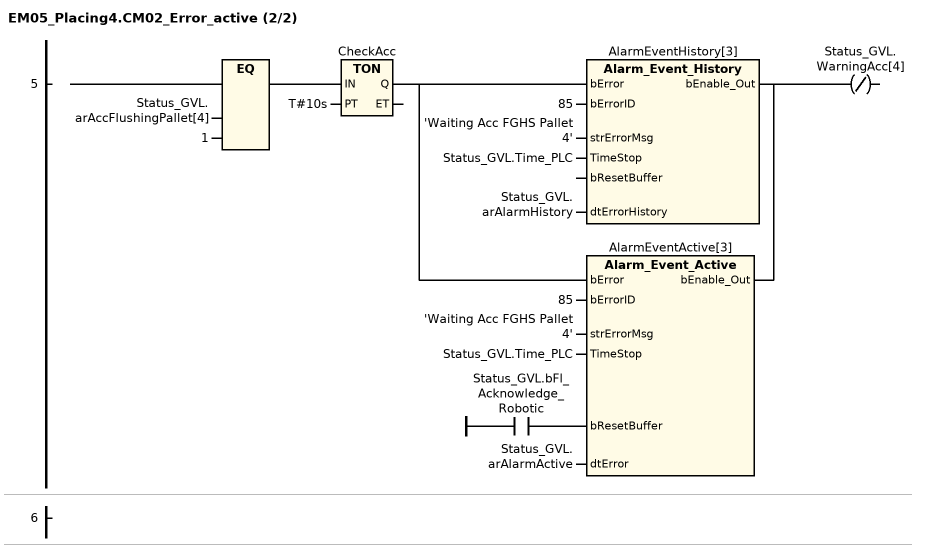
// NETWORK 5
CheckAcc(IN := Status_GVL.arAccFlushingPallet[4] = 1, PT := T#10s); // TON
AlarmEventHistory[3](
    bError := CheckAcc.Q,
    bErrorID := 85,
    strErrorMsg := 'Waiting Acc FGHS Pallet 4',
    TimeStop := Status_GVL.Time_PLC,
    dtErrorHistory := Status_GVL.arAlarmHistory); // Alarm_Event_History
AlarmEventActive[3](
    bError := CheckAcc.Q,
    bErrorID := 85,
    strErrorMsg := 'Waiting Acc FGHS Pallet 4',
    TimeStop := Status_GVL.Time_PLC,
    bResetBuffer := Status_GVL.bFl_Acknowledge_Robotic,
    dtError := Status_GVL.arAlarmActive); // Alarm_Event_Active
Status_GVL.WarningAcc[4] := NOT (AlarmEventHistory[3].bEnable_Out OR AlarmEventActive[3].bEnable_Out);

// NETWORK 6
END_ACTION

ACTION CM03_Output_active:
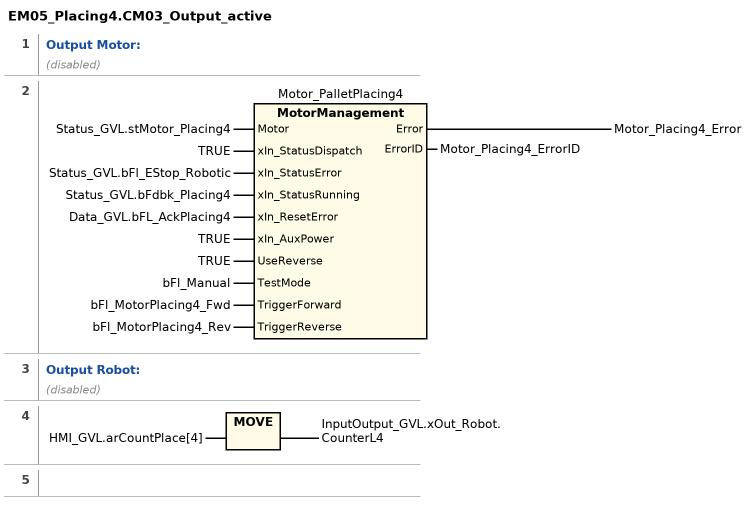
// NETWORK 1 (disabled)
// label: Output Motor

// NETWORK 2
Motor_PalletPlacing4(
    Motor := Status_GVL.stMotor_Placing4,
    xIn_StatusDispatch := TRUE,
    xIn_StatusError := Status_GVL.bFl_EStop_Robotic,
    xIn_StatusRunning := Status_GVL.bFdbk_Placing4,
    xIn_ResetError := Data_GVL.bFL_AckPlacing4,
    xIn_AuxPower := TRUE,
    UseReverse := TRUE,
    TestMode := bFl_Manual,
    TriggerForward := bFl_MotorPlacing4_Fwd,
    TriggerReverse := bFl_MotorPlacing4_Rev,
    ErrorID => Motor_Placing4_ErrorID); // MotorManagement
Motor_Placing4_Error := Motor_PalletPlacing4.Error;

// NETWORK 3 (disabled)
// label: Output Robot

// NETWORK 4
InputOutput_GVL.xOut_Robot.CounterL4 := HMI_GVL.arCountPlace[4];

// NETWORK 5
END_ACTION

ACTION CM04_Running_active:
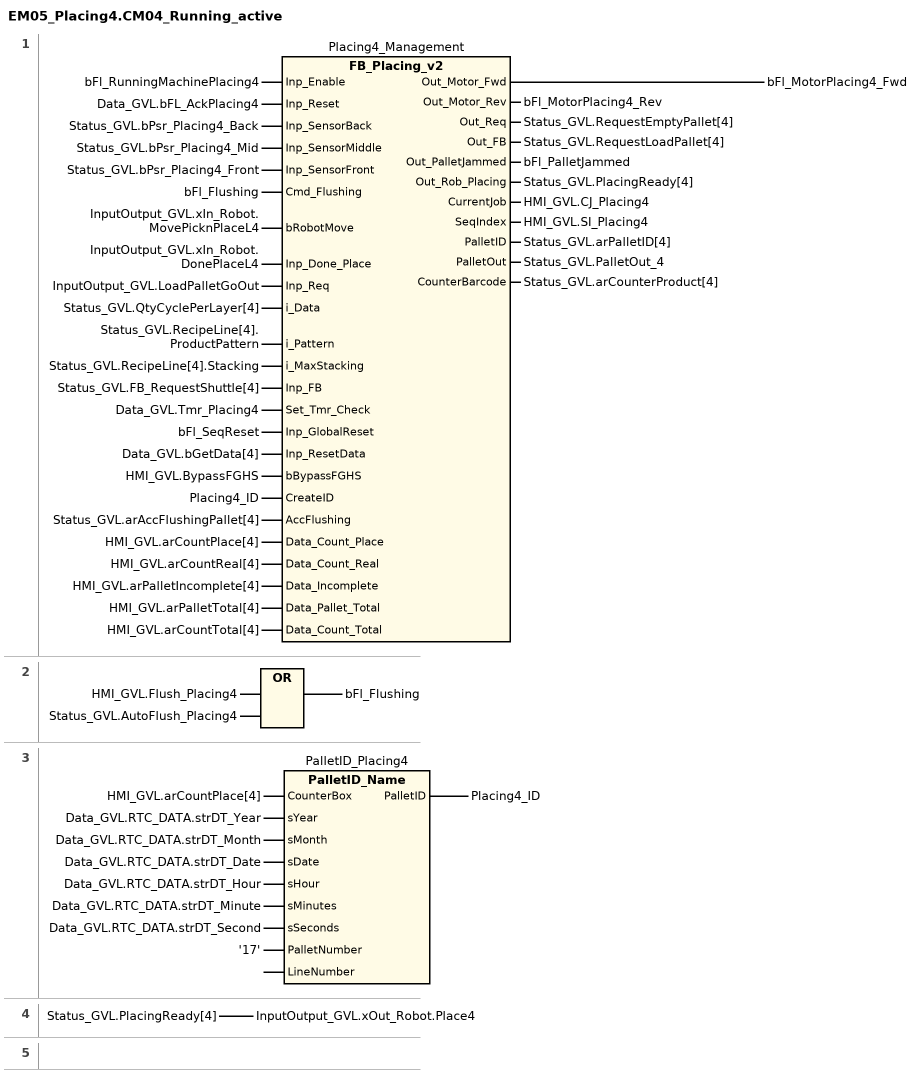
// NETWORK 1
Placing4_Management(
    Inp_Enable := bFl_RunningMachinePlacing4,
    Inp_Reset := Data_GVL.bFL_AckPlacing4,
    Inp_SensorBack := Status_GVL.bPsr_Placing4_Back,
    Inp_SensorMiddle := Status_GVL.bPsr_Placing4_Mid,
    Inp_SensorFront := Status_GVL.bPsr_Placing4_Front,
    Cmd_Flushing := bFl_Flushing,
    bRobotMove := InputOutput_GVL.xIn_Robot.MovePicknPlaceL4,
    Inp_Done_Place := InputOutput_GVL.xIn_Robot.DonePlaceL4,
    Inp_Req := InputOutput_GVL.LoadPalletGoOut,
    i_Data := Status_GVL.QtyCyclePerLayer[4],
    i_Pattern := Status_GVL.RecipeLine[4].ProductPattern,
    i_MaxStacking := Status_GVL.RecipeLine[4].Stacking,
    Inp_FB := Status_GVL.FB_RequestShuttle[4],
    Set_Tmr_Check := Data_GVL.Tmr_Placing4,
    Inp_GlobalReset := bFl_SeqReset,
    Inp_ResetData := Data_GVL.bGetData[4],
    bBypassFGHS := HMI_GVL.BypassFGHS,
    CreateID := Placing4_ID,
    AccFlushing := Status_GVL.arAccFlushingPallet[4],
    Data_Count_Place := HMI_GVL.arCountPlace[4],
    Data_Count_Real := HMI_GVL.arCountReal[4],
    Data_Incomplete := HMI_GVL.arPalletIncomplete[4],
    Data_Pallet_Total := HMI_GVL.arPalletTotal[4],
    Data_Count_Total := HMI_GVL.arCountTotal[4],
    Out_Motor_Rev => bFl_MotorPlacing4_Rev,
    Out_Req => Status_GVL.RequestEmptyPallet[4],
    Out_FB => Status_GVL.RequestLoadPallet[4],
    Out_PalletJammed => bFl_PalletJammed,
    Out_Rob_Placing => Status_GVL.PlacingReady[4],
    CurrentJob => HMI_GVL.CJ_Placing4,
    SeqIndex => HMI_GVL.SI_Placing4,
    PalletID => Status_GVL.arPalletID[4],
    PalletOut => Status_GVL.PalletOut_4,
    CounterBarcode => Status_GVL.arCounterProduct[4]); // FB_Placing_v2
bFl_MotorPlacing4_Fwd := Placing4_Management.Out_Motor_Fwd;

// NETWORK 2
bFl_Flushing := HMI_GVL.Flush_Placing4 OR Status_GVL.AutoFlush_Placing4;

// NETWORK 3
PalletID_Placing4(
    CounterBox := HMI_GVL.arCountPlace[4],
    sYear := Data_GVL.RTC_DATA.strDT_Year,
    sMonth := Data_GVL.RTC_DATA.strDT_Month,
    sDate := Data_GVL.RTC_DATA.strDT_Date,
    sHour := Data_GVL.RTC_DATA.strDT_Hour,
    sMinutes := Data_GVL.RTC_DATA.strDT_Minute,
    sSeconds := Data_GVL.RTC_DATA.strDT_Second,
    PalletNumber := '17'); // PalletID_Name
Placing4_ID := PalletID_Placing4.PalletID;

// NETWORK 4
InputOutput_GVL.xOut_Robot.Place4 := Status_GVL.PlacingReady[4];

// NETWORK 5
END_ACTION

ACTION UP01_Backbone_active:
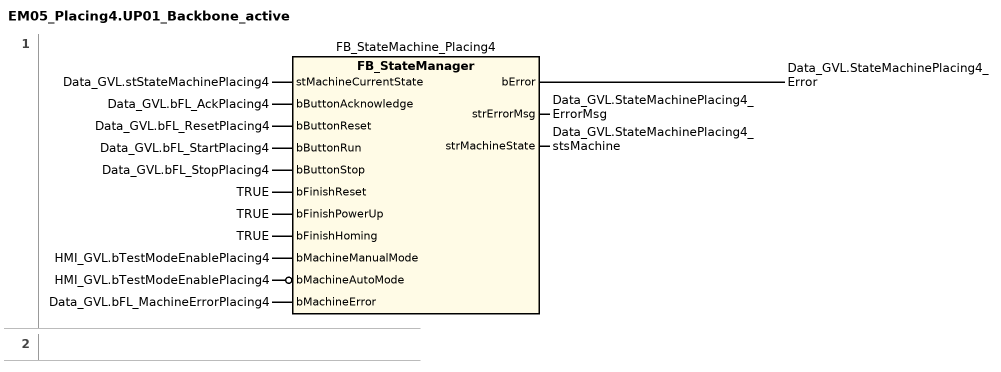
// NETWORK 1
FB_StateMachine_Placing4(
    stMachineCurrentState := Data_GVL.stStateMachinePlacing4,
    bButtonAcknowledge := Data_GVL.bFL_AckPlacing4,
    bButtonReset := Data_GVL.bFL_ResetPlacing4,
    bButtonRun := Data_GVL.bFL_StartPlacing4,
    bButtonStop := Data_GVL.bFL_StopPlacing4,
    bFinishReset := TRUE,
    bFinishPowerUp := TRUE,
    bFinishHoming := TRUE,
    bMachineManualMode := HMI_GVL.bTestModeEnablePlacing4,
    bMachineAutoMode := NOT HMI_GVL.bTestModeEnablePlacing4,
    bMachineError := Data_GVL.bFL_MachineErrorPlacing4,
    strErrorMsg => Data_GVL.StateMachinePlacing4_ErrorMsg,
    strMachineState => Data_GVL.StateMachinePlacing4_stsMachine); // FB_StateManager
Data_GVL.StateMachinePlacing4_Error := FB_StateMachine_Placing4.bError;

// NETWORK 2
END_ACTION

END_PROGRAM

// ---- POUs/S01_Robot/EM06_Picking.TcPOU
PROGRAM EM06_Picking
VAR
	
	//Backbone
	FB_StateMachine_Picking			: FB_StateManager;
	bFl_RunningMachinePicking		: BOOL;
	bFl_SeqReset					: BOOL;
	bFl_Manual						: BOOL;
	CheckStatusPicking				: checkstatus;
	AlarmEventHistory				: ARRAY[1..20] OF Alarm_Event_History;
	ProductFound					: ARRAY [1..4] OF BOOL;
	
	//Motor
	Motor_BoxPicking				: MotorManagement;
	bFl_MotorPicking				: BOOL;
	Motor_Picking_Error				: BOOL;
	Motor_Picking_ErrorID			: UINT;
	
	//Pneumatic
	Pneumatic_GapMaker				: Pneumatic_2Coil_Management;
	bFl_GapMaker_Rtc				: BOOL;
	bFl_GapMaker_Adv				: BOOL;
	Pneu_GapMaker_Error				: BOOL;	
	Pneu_GapMaker_ErrorMsg			: STRING;
	
	Pneumatic_Centering				: Pneumatic_1Coil_Management;
	bFl_Centering					: BOOL;
	Pneu_Centering_Error			: BOOL;	
	Pneu_Centering_ErrorMsg			: STRING;
	
	//Picking
	Picking							: FB_Picking;
	
	//Barcode Reader
	bFl_BarcodeChecked				: BOOL;
	bFl_TriggerBarcode				: BOOL;
	bFl_DoneRead_Barcode_Picking	: ARRAY [1..4] OF BOOL;
	bFl_GoodRead_Barcode_Picking	: ARRAY [1..4] OF BOOL;
	bFl_BadRead_Barcode_Picking		: ARRAY [1..4] OF BOOL;
	BarcodeInspection				: FB_BarcodeInspection;
	BarcodeReader_Picking1			: DM_Connect;
	BarcodeReader_Picking2			: DM_Connect;
	BarcodeReader_Picking3			: DM_Connect;
	BarcodeReader_Picking4			: DM_Connect;
	DataBarcode_Picking1			: STRING;
	DataBarcode_Picking2			: STRING;
	DataBarcode_Picking3			: STRING;
	DataBarcode_Picking4			: STRING;
	Barcode1_Error					: BOOL;
	Barcode2_Error					: BOOL;
	Barcode3_Error					: BOOL;
	Barcode4_Error					: BOOL;
	TestRun							: BOOL;
	TestTrigger						: BOOL;
	LEN1							: INT;
	POS1							: INT;
	POS2							: INT;
	LEN_2							: INT;
	LinkUp							: STRING(255);
	RotatePicking					: RotatePick;
	DonePick						: BOOL;
	bFL_Safety						: BOOL;
	AutoReset						: BOOL;
	TON_Auto						: TON;
	AutoAck							: BOOL;
	AutoRun							: BOOL;
	TOF_Run							: TOF;
	TOF_Reset						: TOF;
	AlarmEventActive				: ARRAY[1..20] OF Alarm_Event_Active;
	RejectMsgList					: RejectMsgHandling;
	bReject							: BOOL;
	RejectID						: INT;
	RejectMsg						: STRING;
	CounterReject					: UINT;
	bRotate							: BOOL;
	BarcodeReader_Picking2B			: DM_Connect;
	Barcode2B_Error					: BOOL;
	DataBarcode_Picking2B			: STRING;
	bFl_DoneRead_Barcode_Picking2B	: BOOL;
	
	BarcodeReader_Picking3B			: DM_Connect;
	Barcode3B_Error					: BOOL;
	DataBarcode_Picking3B			: STRING;
	intRotatePick					: USINT;
END_VAR
VAR // added by the converter: edge detectors and wires of the graphical bodies
    _w1 : BOOL;
END_VAR

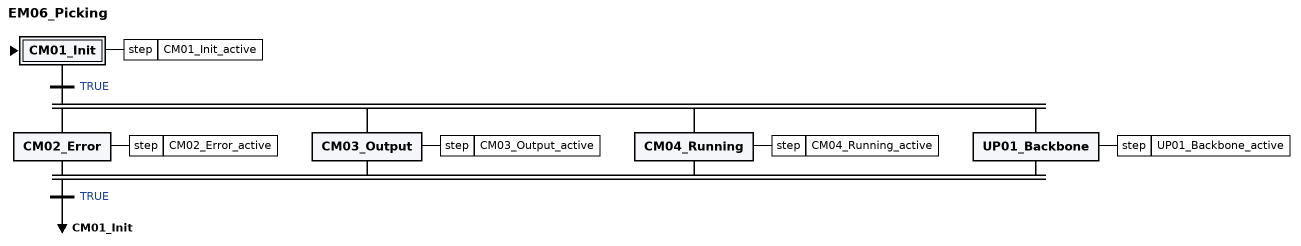
INITIAL_STEP CM01_Init:
    CM01_Init_active(N);  // step action
END_STEP
TRANSITION FROM CM01_Init TO (CM02_Error, CM03_Output, CM04_Running, UP01_Backbone)
    := TRUE;
END_TRANSITION
STEP CM02_Error:
    CM02_Error_active(N);  // step action
END_STEP
STEP CM03_Output:
    CM03_Output_active(N);  // step action
END_STEP
STEP CM04_Running:
    CM04_Running_active(N);  // step action
END_STEP
STEP UP01_Backbone:
    UP01_Backbone_active(N);  // step action
END_STEP
TRANSITION FROM (CM02_Error, CM03_Output, CM04_Running, UP01_Backbone) TO CM01_Init
    := TRUE;
END_TRANSITION

ACTION CM01_Init_active:
Data_GVL.bFL_StartPicking			:= Status_GVL.bFl_RunButton_Robotic OR HMI_GVL.bStartButtonPicking OR HMI_GVL.bAutoStartPicking;
Data_GVL.bFL_StopPicking			:= NOT Status_GVL.bFl_StopButton_Robotic OR HMI_GVL.bStopButtonPicking;
Data_GVL.bFL_ResetPicking			:= Status_GVL.bFl_ResetButton_Robotic OR HMI_GVL.bResetButtonPicking OR HMI_GVL.bAutoResetPicking;
Data_GVL.bFL_AckPicking				:= Status_GVL.bFl_Acknowledge_Robotic OR HMI_GVL.bAcknowledgeButtonPicking OR HMI_GVL.bAutoAcknowledgePicking;
Data_GVL.bFL_AutoManuaModePicking 	:= Status_GVL.bFl_Manual_Robotic OR HMI_GVL.bTestModeEnablePicking;
bFl_RunningMachinePicking			:= Data_GVL.stStateMachinePicking.Running;
bFl_Manual							:= Data_GVL.stStateMachinePicking.ManualMode;
bFl_SeqReset						:= NOT Status_GVL.bFl_EStop_Robotic;
bFL_Safety							:= Status_GVL.bFl_EStop_Robotic AND Status_GVL.bSafety_DoorRobotic AND Status_GVL.bAirPressure_Robotic;



(*=================Convert Timer============================*)
Data_GVL.Tmr_Picking	:= ConvertMilliSecTimeData(HMI_GVL.Tmr_Picking);
Data_GVL.Tmr_Centering	:= ConvertMilliSecTimeData(HMI_GVL.Tmr_Centering);

(*=================Auto Flushing============================*)
//Place1
IF ProductFound[1] AND HMI_GVL.arCountReal[1] > 1 THEN
	Status_GVL.AutoFlush_Placing1	:= TRUE;
ELSE
	Status_GVL.AutoFlush_Placing1	:= FALSE;
END_IF

//Place2
IF ProductFound[2] AND HMI_GVL.arCountReal[2] > 1 THEN
	Status_GVL.AutoFlush_Placing2	:= TRUE;
ELSE
	Status_GVL.AutoFlush_Placing2	:= FALSE;
END_IF

//Place3
IF ProductFound[3] AND HMI_GVL.arCountReal[3] > 1 THEN
	Status_GVL.AutoFlush_Placing3	:= TRUE;
ELSE
	Status_GVL.AutoFlush_Placing3	:= FALSE;
END_IF

//Place4
IF ProductFound[4] AND HMI_GVL.arCountReal[4] > 1 THEN
	Status_GVL.AutoFlush_Placing4	:= TRUE;
ELSE
	Status_GVL.AutoFlush_Placing4	:= FALSE;
END_IF
END_ACTION

ACTION CM02_Error_active:
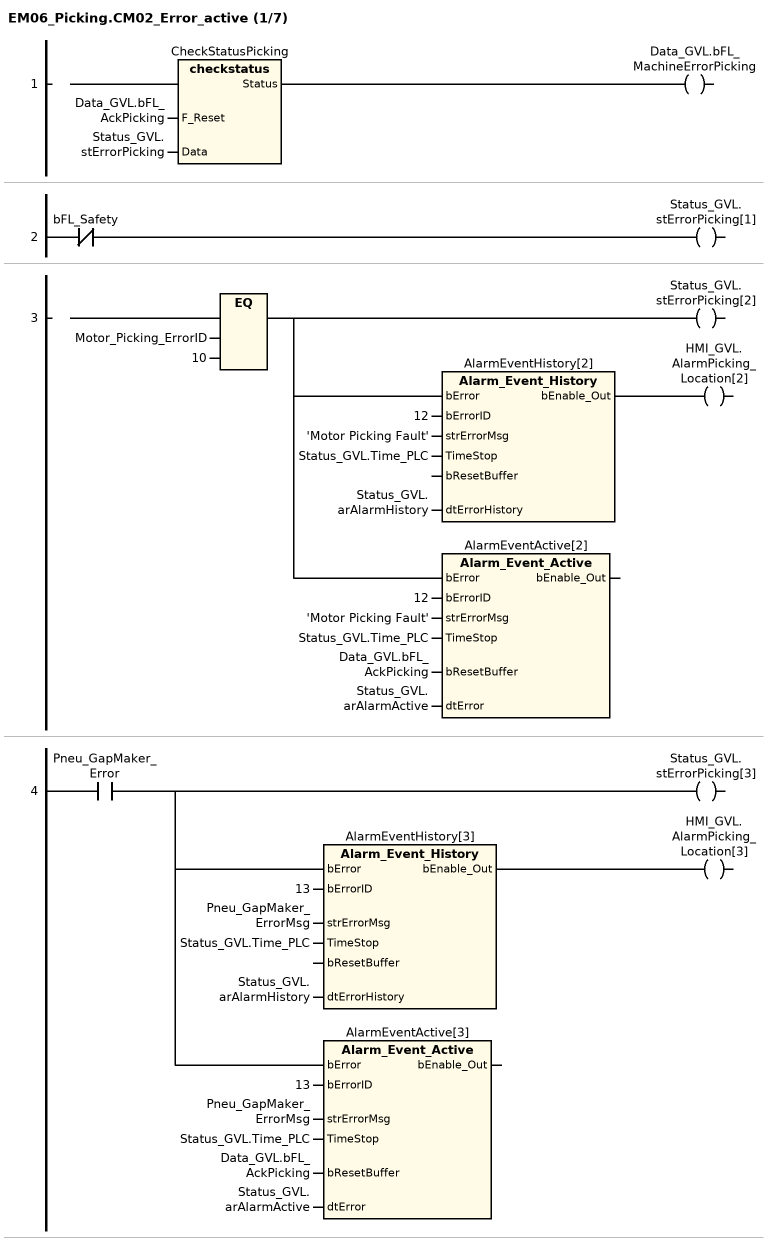
// NETWORK 1
CheckStatusPicking(F_Reset := Data_GVL.bFL_AckPicking, Data := Status_GVL.stErrorPicking); // checkstatus
Data_GVL.bFL_MachineErrorPicking := CheckStatusPicking.Status;

// NETWORK 2
Status_GVL.stErrorPicking[1] := NOT bFL_Safety;

// NETWORK 3
_w1 := Motor_Picking_ErrorID = 10;
Status_GVL.stErrorPicking[2] := _w1;
AlarmEventHistory[2](
    bError := _w1,
    bErrorID := 12,
    strErrorMsg := 'Motor Picking Fault',
    TimeStop := Status_GVL.Time_PLC,
    dtErrorHistory := Status_GVL.arAlarmHistory); // Alarm_Event_History
HMI_GVL.AlarmPicking_Location[2] := AlarmEventHistory[2].bEnable_Out;
AlarmEventActive[2](
    bError := _w1,
    bErrorID := 12,
    strErrorMsg := 'Motor Picking Fault',
    TimeStop := Status_GVL.Time_PLC,
    bResetBuffer := Data_GVL.bFL_AckPicking,
    dtError := Status_GVL.arAlarmActive); // Alarm_Event_Active

// NETWORK 4
Status_GVL.stErrorPicking[3] := Pneu_GapMaker_Error;
AlarmEventHistory[3](
    bError := Pneu_GapMaker_Error,
    bErrorID := 13,
    strErrorMsg := Pneu_GapMaker_ErrorMsg,
    TimeStop := Status_GVL.Time_PLC,
    dtErrorHistory := Status_GVL.arAlarmHistory); // Alarm_Event_History
HMI_GVL.AlarmPicking_Location[3] := AlarmEventHistory[3].bEnable_Out;
AlarmEventActive[3](
    bError := Pneu_GapMaker_Error,
    bErrorID := 13,
    strErrorMsg := Pneu_GapMaker_ErrorMsg,
    TimeStop := Status_GVL.Time_PLC,
    bResetBuffer := Data_GVL.bFL_AckPicking,
    dtError := Status_GVL.arAlarmActive); // Alarm_Event_Active

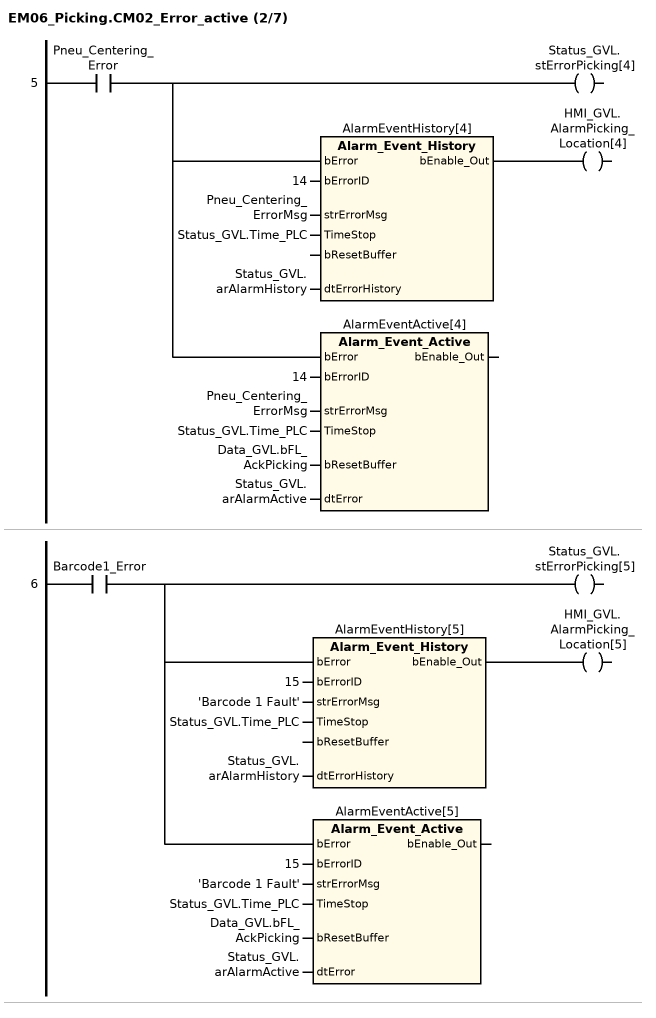
// NETWORK 5
Status_GVL.stErrorPicking[4] := Pneu_Centering_Error;
AlarmEventHistory[4](
    bError := Pneu_Centering_Error,
    bErrorID := 14,
    strErrorMsg := Pneu_Centering_ErrorMsg,
    TimeStop := Status_GVL.Time_PLC,
    dtErrorHistory := Status_GVL.arAlarmHistory); // Alarm_Event_History
HMI_GVL.AlarmPicking_Location[4] := AlarmEventHistory[4].bEnable_Out;
AlarmEventActive[4](
    bError := Pneu_Centering_Error,
    bErrorID := 14,
    strErrorMsg := Pneu_Centering_ErrorMsg,
    TimeStop := Status_GVL.Time_PLC,
    bResetBuffer := Data_GVL.bFL_AckPicking,
    dtError := Status_GVL.arAlarmActive); // Alarm_Event_Active

// NETWORK 6
Status_GVL.stErrorPicking[5] := Barcode1_Error;
AlarmEventHistory[5](
    bError := Barcode1_Error,
    bErrorID := 15,
    strErrorMsg := 'Barcode 1 Fault',
    TimeStop := Status_GVL.Time_PLC,
    dtErrorHistory := Status_GVL.arAlarmHistory); // Alarm_Event_History
HMI_GVL.AlarmPicking_Location[5] := AlarmEventHistory[5].bEnable_Out;
AlarmEventActive[5](
    bError := Barcode1_Error,
    bErrorID := 15,
    strErrorMsg := 'Barcode 1 Fault',
    TimeStop := Status_GVL.Time_PLC,
    bResetBuffer := Data_GVL.bFL_AckPicking,
    dtError := Status_GVL.arAlarmActive); // Alarm_Event_Active

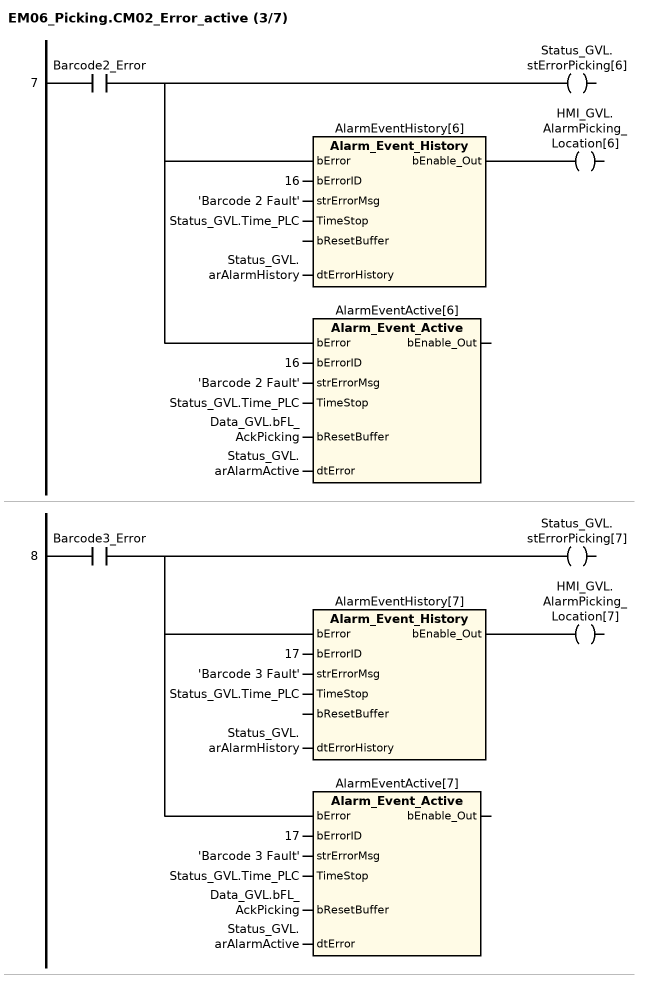
// NETWORK 7
Status_GVL.stErrorPicking[6] := Barcode2_Error;
AlarmEventHistory[6](
    bError := Barcode2_Error,
    bErrorID := 16,
    strErrorMsg := 'Barcode 2 Fault',
    TimeStop := Status_GVL.Time_PLC,
    dtErrorHistory := Status_GVL.arAlarmHistory); // Alarm_Event_History
HMI_GVL.AlarmPicking_Location[6] := AlarmEventHistory[6].bEnable_Out;
AlarmEventActive[6](
    bError := Barcode2_Error,
    bErrorID := 16,
    strErrorMsg := 'Barcode 2 Fault',
    TimeStop := Status_GVL.Time_PLC,
    bResetBuffer := Data_GVL.bFL_AckPicking,
    dtError := Status_GVL.arAlarmActive); // Alarm_Event_Active

// NETWORK 8
Status_GVL.stErrorPicking[7] := Barcode3_Error;
AlarmEventHistory[7](
    bError := Barcode3_Error,
    bErrorID := 17,
    strErrorMsg := 'Barcode 3 Fault',
    TimeStop := Status_GVL.Time_PLC,
    dtErrorHistory := Status_GVL.arAlarmHistory); // Alarm_Event_History
HMI_GVL.AlarmPicking_Location[7] := AlarmEventHistory[7].bEnable_Out;
AlarmEventActive[7](
    bError := Barcode3_Error,
    bErrorID := 17,
    strErrorMsg := 'Barcode 3 Fault',
    TimeStop := Status_GVL.Time_PLC,
    bResetBuffer := Data_GVL.bFL_AckPicking,
    dtError := Status_GVL.arAlarmActive); // Alarm_Event_Active

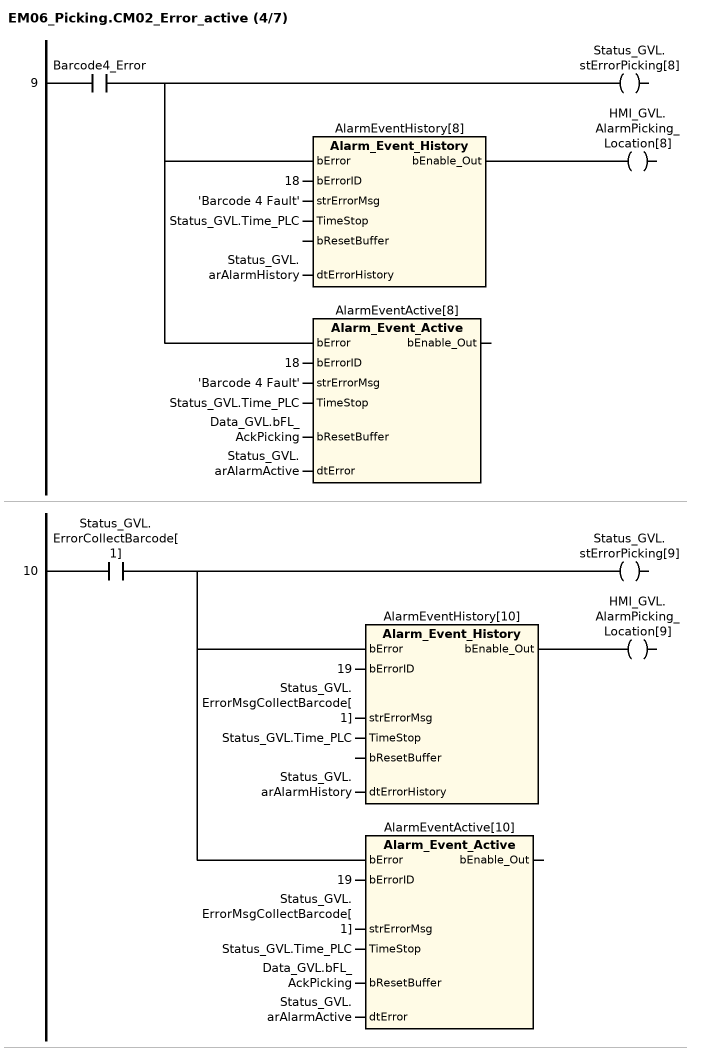
// NETWORK 9
Status_GVL.stErrorPicking[8] := Barcode4_Error;
AlarmEventHistory[8](
    bError := Barcode4_Error,
    bErrorID := 18,
    strErrorMsg := 'Barcode 4 Fault',
    TimeStop := Status_GVL.Time_PLC,
    dtErrorHistory := Status_GVL.arAlarmHistory); // Alarm_Event_History
HMI_GVL.AlarmPicking_Location[8] := AlarmEventHistory[8].bEnable_Out;
AlarmEventActive[8](
    bError := Barcode4_Error,
    bErrorID := 18,
    strErrorMsg := 'Barcode 4 Fault',
    TimeStop := Status_GVL.Time_PLC,
    bResetBuffer := Data_GVL.bFL_AckPicking,
    dtError := Status_GVL.arAlarmActive); // Alarm_Event_Active

// NETWORK 10
Status_GVL.stErrorPicking[9] := Status_GVL.ErrorCollectBarcode[1];
AlarmEventHistory[10](
    bError := Status_GVL.ErrorCollectBarcode[1],
    bErrorID := 19,
    strErrorMsg := Status_GVL.ErrorMsgCollectBarcode[1],
    TimeStop := Status_GVL.Time_PLC,
    dtErrorHistory := Status_GVL.arAlarmHistory); // Alarm_Event_History
HMI_GVL.AlarmPicking_Location[9] := AlarmEventHistory[10].bEnable_Out;
AlarmEventActive[10](
    bError := Status_GVL.ErrorCollectBarcode[1],
    bErrorID := 19,
    strErrorMsg := Status_GVL.ErrorMsgCollectBarcode[1],
    TimeStop := Status_GVL.Time_PLC,
    bResetBuffer := Data_GVL.bFL_AckPicking,
    dtError := Status_GVL.arAlarmActive); // Alarm_Event_Active

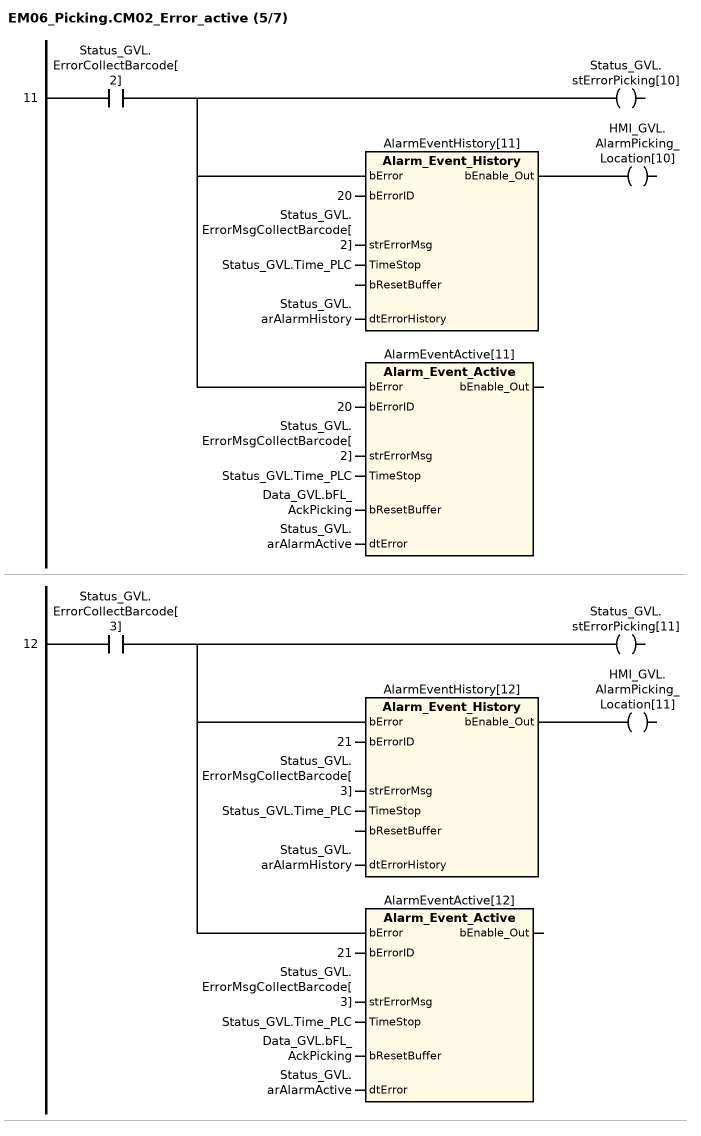
// NETWORK 11
Status_GVL.stErrorPicking[10] := Status_GVL.ErrorCollectBarcode[2];
AlarmEventHistory[11](
    bError := Status_GVL.ErrorCollectBarcode[2],
    bErrorID := 20,
    strErrorMsg := Status_GVL.ErrorMsgCollectBarcode[2],
    TimeStop := Status_GVL.Time_PLC,
    dtErrorHistory := Status_GVL.arAlarmHistory); // Alarm_Event_History
HMI_GVL.AlarmPicking_Location[10] := AlarmEventHistory[11].bEnable_Out;
AlarmEventActive[11](
    bError := Status_GVL.ErrorCollectBarcode[2],
    bErrorID := 20,
    strErrorMsg := Status_GVL.ErrorMsgCollectBarcode[2],
    TimeStop := Status_GVL.Time_PLC,
    bResetBuffer := Data_GVL.bFL_AckPicking,
    dtError := Status_GVL.arAlarmActive); // Alarm_Event_Active

// NETWORK 12
Status_GVL.stErrorPicking[11] := Status_GVL.ErrorCollectBarcode[3];
AlarmEventHistory[12](
    bError := Status_GVL.ErrorCollectBarcode[3],
    bErrorID := 21,
    strErrorMsg := Status_GVL.ErrorMsgCollectBarcode[3],
    TimeStop := Status_GVL.Time_PLC,
    dtErrorHistory := Status_GVL.arAlarmHistory); // Alarm_Event_History
HMI_GVL.AlarmPicking_Location[11] := AlarmEventHistory[12].bEnable_Out;
AlarmEventActive[12](
    bError := Status_GVL.ErrorCollectBarcode[3],
    bErrorID := 21,
    strErrorMsg := Status_GVL.ErrorMsgCollectBarcode[3],
    TimeStop := Status_GVL.Time_PLC,
    bResetBuffer := Data_GVL.bFL_AckPicking,
    dtError := Status_GVL.arAlarmActive); // Alarm_Event_Active

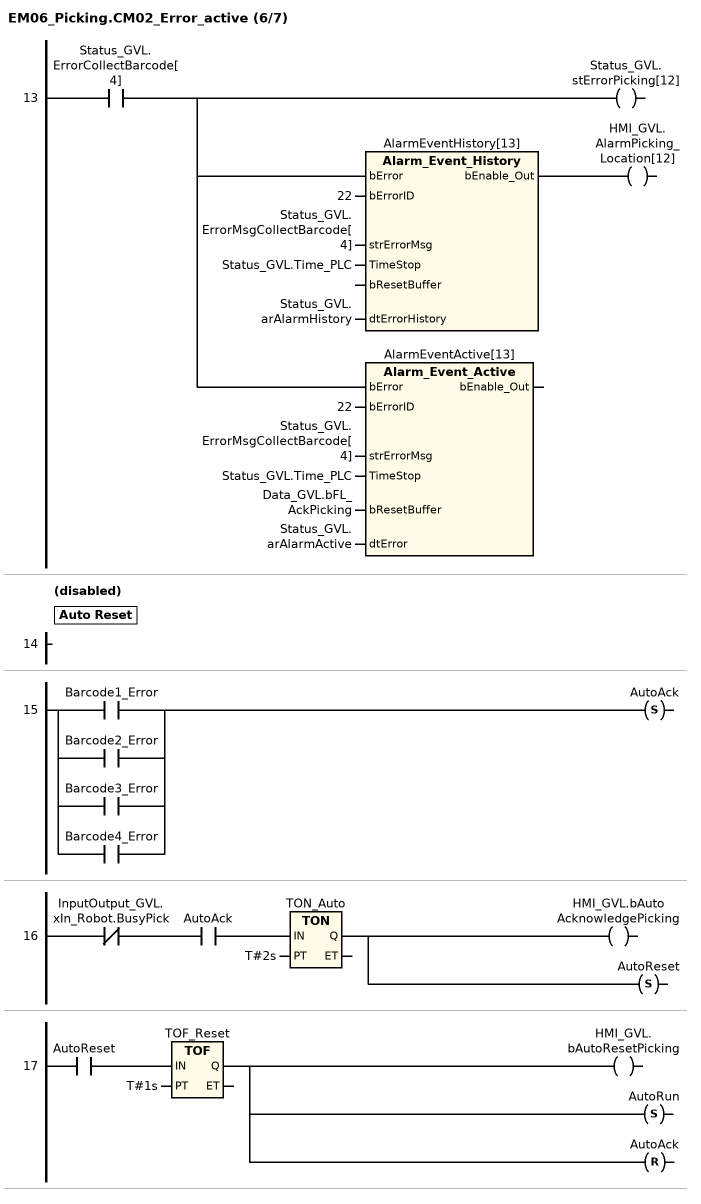
// NETWORK 13
Status_GVL.stErrorPicking[12] := Status_GVL.ErrorCollectBarcode[4];
AlarmEventHistory[13](
    bError := Status_GVL.ErrorCollectBarcode[4],
    bErrorID := 22,
    strErrorMsg := Status_GVL.ErrorMsgCollectBarcode[4],
    TimeStop := Status_GVL.Time_PLC,
    dtErrorHistory := Status_GVL.arAlarmHistory); // Alarm_Event_History
HMI_GVL.AlarmPicking_Location[12] := AlarmEventHistory[13].bEnable_Out;
AlarmEventActive[13](
    bError := Status_GVL.ErrorCollectBarcode[4],
    bErrorID := 22,
    strErrorMsg := Status_GVL.ErrorMsgCollectBarcode[4],
    TimeStop := Status_GVL.Time_PLC,
    bResetBuffer := Data_GVL.bFL_AckPicking,
    dtError := Status_GVL.arAlarmActive); // Alarm_Event_Active

// NETWORK 14 (disabled)
// label: Auto Reset

// NETWORK 15
AutoAck S= Barcode1_Error OR Barcode2_Error OR Barcode3_Error OR Barcode4_Error;

// NETWORK 16
TON_Auto(IN := NOT InputOutput_GVL.xIn_Robot.BusyPick AND AutoAck, PT := T#2s); // TON
HMI_GVL.bAutoAcknowledgePicking := TON_Auto.Q;
AutoReset S= TON_Auto.Q;

// NETWORK 17
TOF_Reset(IN := AutoReset, PT := T#1s); // TOF
HMI_GVL.bAutoResetPicking := TOF_Reset.Q;
AutoRun S= TOF_Reset.Q;
AutoAck R= TOF_Reset.Q;

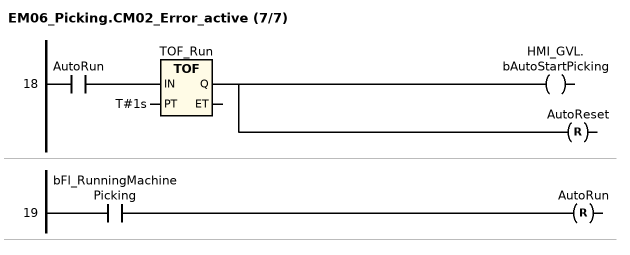
// NETWORK 18
TOF_Run(IN := AutoRun, PT := T#1s); // TOF
HMI_GVL.bAutoStartPicking := TOF_Run.Q;
AutoReset R= TOF_Run.Q;

// NETWORK 19
AutoRun R= bFl_RunningMachinePicking;
END_ACTION

ACTION CM03_Output_active:
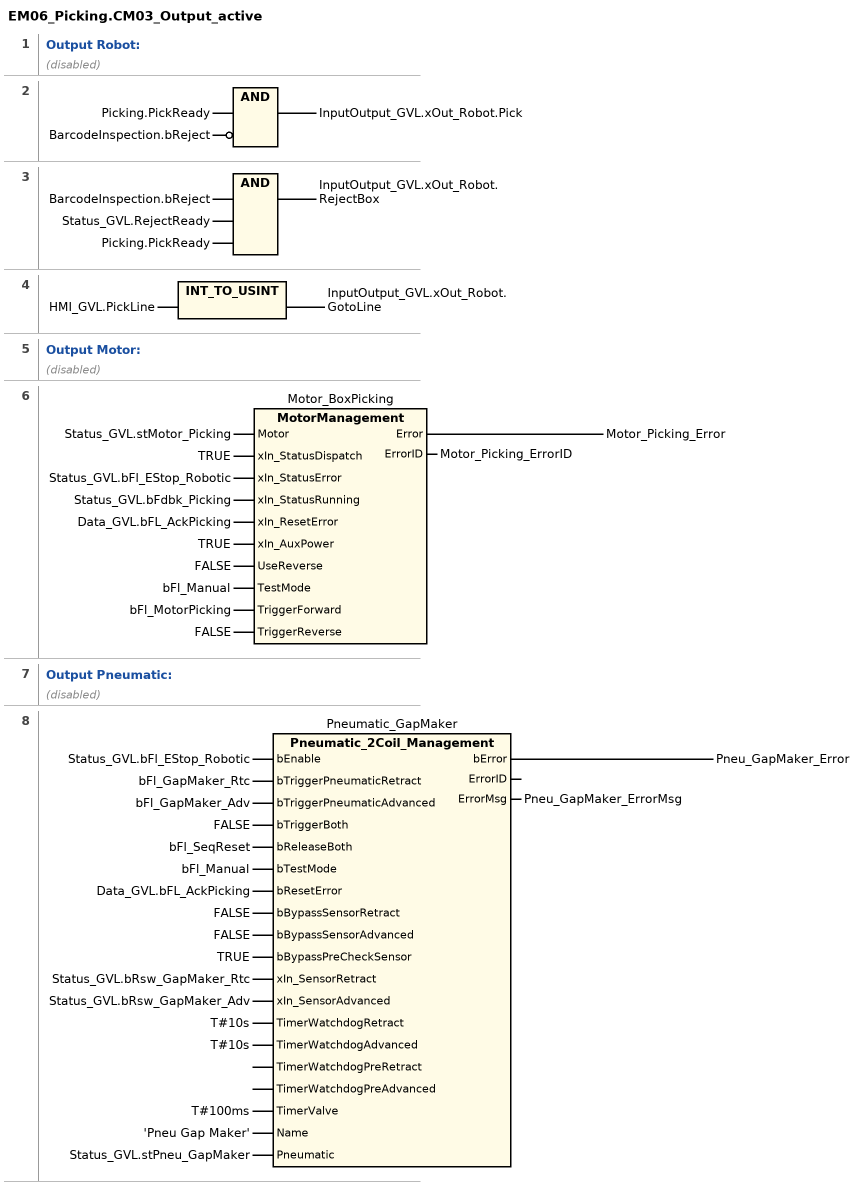
// NETWORK 1 (disabled)
// label: Output Robot

// NETWORK 2
InputOutput_GVL.xOut_Robot.Pick := Picking.PickReady AND NOT BarcodeInspection.bReject;

// NETWORK 3
InputOutput_GVL.xOut_Robot.RejectBox := BarcodeInspection.bReject AND Status_GVL.RejectReady AND Picking.PickReady;

// NETWORK 4
InputOutput_GVL.xOut_Robot.GotoLine := INT_TO_USINT(HMI_GVL.PickLine);

// NETWORK 5 (disabled)
// label: Output Motor

// NETWORK 6
Motor_BoxPicking(
    Motor := Status_GVL.stMotor_Picking,
    xIn_StatusDispatch := TRUE,
    xIn_StatusError := Status_GVL.bFl_EStop_Robotic,
    xIn_StatusRunning := Status_GVL.bFdbk_Picking,
    xIn_ResetError := Data_GVL.bFL_AckPicking,
    xIn_AuxPower := TRUE,
    UseReverse := FALSE,
    TestMode := bFl_Manual,
    TriggerForward := bFl_MotorPicking,
    TriggerReverse := FALSE,
    ErrorID => Motor_Picking_ErrorID); // MotorManagement
Motor_Picking_Error := Motor_BoxPicking.Error;

// NETWORK 7 (disabled)
// label: Output Pneumatic

// NETWORK 8
Pneumatic_GapMaker(
    bEnable := Status_GVL.bFl_EStop_Robotic,
    bTriggerPneumaticRetract := bFl_GapMaker_Rtc,
    bTriggerPneumaticAdvanced := bFl_GapMaker_Adv,
    bTriggerBoth := FALSE,
    bReleaseBoth := bFl_SeqReset,
    bTestMode := bFl_Manual,
    bResetError := Data_GVL.bFL_AckPicking,
    bBypassSensorRetract := FALSE,
    bBypassSensorAdvanced := FALSE,
    bBypassPreCheckSensor := TRUE,
    xIn_SensorRetract := Status_GVL.bRsw_GapMaker_Rtc,
    xIn_SensorAdvanced := Status_GVL.bRsw_GapMaker_Adv,
    TimerWatchdogRetract := T#10s,
    TimerWatchdogAdvanced := T#10s,
    TimerValve := T#100ms,
    Name := 'Pneu Gap Maker',
    Pneumatic := Status_GVL.stPneu_GapMaker,
    ErrorMsg => Pneu_GapMaker_ErrorMsg); // Pneumatic_2Coil_Management
Pneu_GapMaker_Error := Pneumatic_GapMaker.bError;

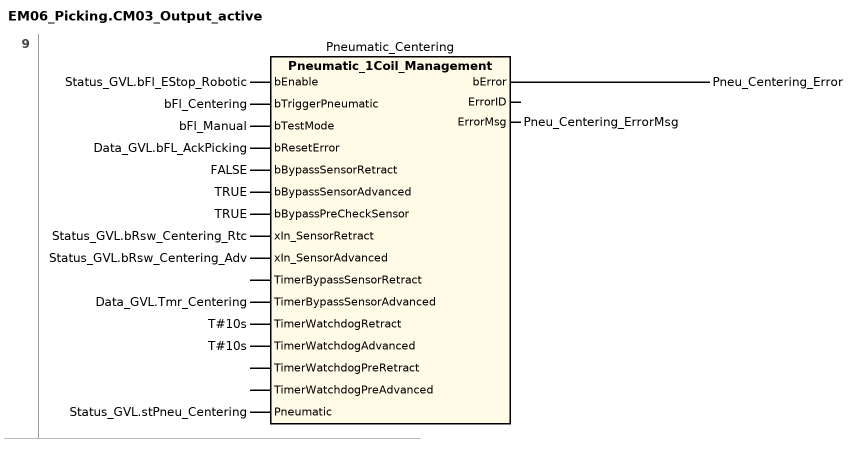
// NETWORK 9
Pneumatic_Centering(
    bEnable := Status_GVL.bFl_EStop_Robotic,
    bTriggerPneumatic := bFl_Centering,
    bTestMode := bFl_Manual,
    bResetError := Data_GVL.bFL_AckPicking,
    bBypassSensorRetract := FALSE,
    bBypassSensorAdvanced := TRUE,
    bBypassPreCheckSensor := TRUE,
    xIn_SensorRetract := Status_GVL.bRsw_Centering_Rtc,
    xIn_SensorAdvanced := Status_GVL.bRsw_Centering_Adv,
    TimerBypassSensorAdvanced := Data_GVL.Tmr_Centering,
    TimerWatchdogRetract := T#10s,
    TimerWatchdogAdvanced := T#10s,
    Pneumatic := Status_GVL.stPneu_Centering,
    ErrorMsg => Pneu_Centering_ErrorMsg); // Pneumatic_1Coil_Management
Pneu_Centering_Error := Pneumatic_Centering.bError;
END_ACTION

ACTION CM04_Running_active:
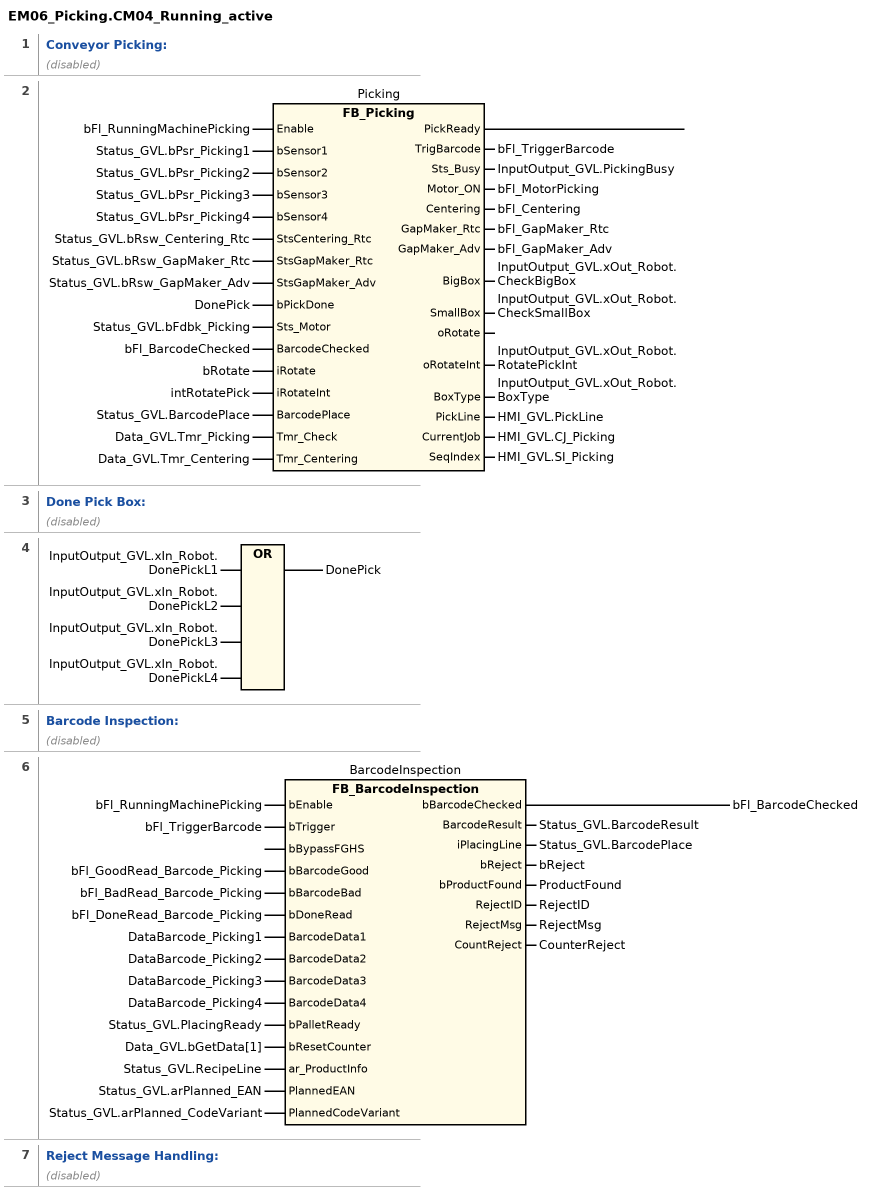
// NETWORK 1 (disabled)
// label: Conveyor Picking

// NETWORK 2
Picking(
    Enable := bFl_RunningMachinePicking,
    bSensor1 := Status_GVL.bPsr_Picking1,
    bSensor2 := Status_GVL.bPsr_Picking2,
    bSensor3 := Status_GVL.bPsr_Picking3,
    bSensor4 := Status_GVL.bPsr_Picking4,
    StsCentering_Rtc := Status_GVL.bRsw_Centering_Rtc,
    StsGapMaker_Rtc := Status_GVL.bRsw_GapMaker_Rtc,
    StsGapMaker_Adv := Status_GVL.bRsw_GapMaker_Adv,
    bPickDone := DonePick,
    Sts_Motor := Status_GVL.bFdbk_Picking,
    BarcodeChecked := bFl_BarcodeChecked,
    iRotate := bRotate,
    iRotateInt := intRotatePick,
    BarcodePlace := Status_GVL.BarcodePlace,
    Tmr_Check := Data_GVL.Tmr_Picking,
    Tmr_Centering := Data_GVL.Tmr_Centering,
    TrigBarcode => bFl_TriggerBarcode,
    Sts_Busy => InputOutput_GVL.PickingBusy,
    Motor_ON => bFl_MotorPicking,
    Centering => bFl_Centering,
    GapMaker_Rtc => bFl_GapMaker_Rtc,
    GapMaker_Adv => bFl_GapMaker_Adv,
    BigBox => InputOutput_GVL.xOut_Robot.CheckBigBox,
    SmallBox => InputOutput_GVL.xOut_Robot.CheckSmallBox,
    oRotateInt => InputOutput_GVL.xOut_Robot.RotatePickInt,
    BoxType => InputOutput_GVL.xOut_Robot.BoxType,
    PickLine => HMI_GVL.PickLine,
    CurrentJob => HMI_GVL.CJ_Picking,
    SeqIndex => HMI_GVL.SI_Picking); // FB_Picking

// NETWORK 3 (disabled)
// label: Done Pick Box

// NETWORK 4
DonePick := InputOutput_GVL.xIn_Robot.DonePickL1 OR InputOutput_GVL.xIn_Robot.DonePickL2 OR InputOutput_GVL.xIn_Robot.DonePickL3 OR InputOutput_GVL.xIn_Robot.DonePickL4;

// NETWORK 5 (disabled)
// label: Barcode Inspection

// NETWORK 6
BarcodeInspection(
    bEnable := bFl_RunningMachinePicking,
    bTrigger := bFl_TriggerBarcode,
    bBarcodeGood := bFl_GoodRead_Barcode_Picking,
    bBarcodeBad := bFl_BadRead_Barcode_Picking,
    bDoneRead := bFl_DoneRead_Barcode_Picking,
    BarcodeData1 := DataBarcode_Picking1,
    BarcodeData2 := DataBarcode_Picking2,
    BarcodeData3 := DataBarcode_Picking3,
    BarcodeData4 := DataBarcode_Picking4,
    bPalletReady := Status_GVL.PlacingReady,
    bResetCounter := Data_GVL.bGetData[1],
    ar_ProductInfo := Status_GVL.RecipeLine,
    PlannedEAN := Status_GVL.arPlanned_EAN,
    PlannedCodeVariant := Status_GVL.arPlanned_CodeVariant,
    BarcodeResult => Status_GVL.BarcodeResult,
    iPlacingLine => Status_GVL.BarcodePlace,
    bReject => bReject,
    bProductFound => ProductFound,
    RejectID => RejectID,
    RejectMsg => RejectMsg,
    CountReject => CounterReject); // FB_BarcodeInspection
bFl_BarcodeChecked := BarcodeInspection.bBarcodeChecked;

// NETWORK 7 (disabled)
// label: Reject Message Handling

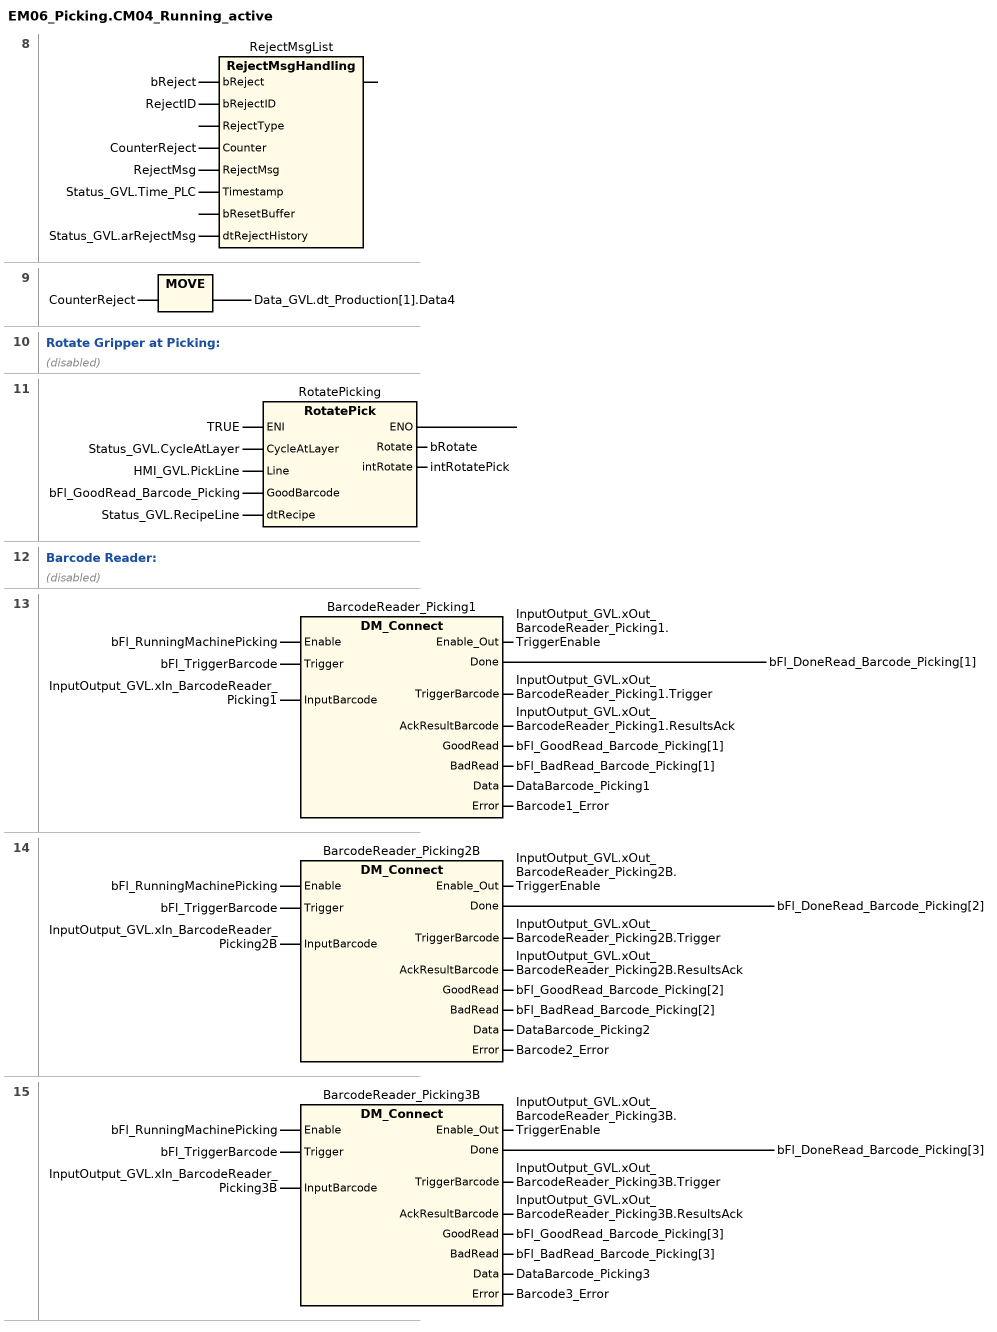
// NETWORK 8
RejectMsgList(
    bReject := bReject,
    bRejectID := RejectID,
    Counter := CounterReject,
    RejectMsg := RejectMsg,
    Timestamp := Status_GVL.Time_PLC,
    dtRejectHistory := Status_GVL.arRejectMsg); // RejectMsgHandling

// NETWORK 9
Data_GVL.dt_Production[1].Data4 := CounterReject;

// NETWORK 10 (disabled)
// label: Rotate Gripper at Picking

// NETWORK 11
RotatePicking(
    ENI := TRUE,
    CycleAtLayer := Status_GVL.CycleAtLayer,
    Line := HMI_GVL.PickLine,
    GoodBarcode := bFl_GoodRead_Barcode_Picking,
    dtRecipe := Status_GVL.RecipeLine,
    Rotate => bRotate,
    intRotate => intRotatePick); // RotatePick

// NETWORK 12 (disabled)
// label: Barcode Reader

// NETWORK 13
BarcodeReader_Picking1(
    Enable := bFl_RunningMachinePicking,
    Trigger := bFl_TriggerBarcode,
    InputBarcode := InputOutput_GVL.xIn_BarcodeReader_Picking1,
    Enable_Out => InputOutput_GVL.xOut_BarcodeReader_Picking1.TriggerEnable,
    TriggerBarcode => InputOutput_GVL.xOut_BarcodeReader_Picking1.Trigger,
    AckResultBarcode => InputOutput_GVL.xOut_BarcodeReader_Picking1.ResultsAck,
    GoodRead => bFl_GoodRead_Barcode_Picking[1],
    BadRead => bFl_BadRead_Barcode_Picking[1],
    Data => DataBarcode_Picking1,
    Error => Barcode1_Error); // DM_Connect
bFl_DoneRead_Barcode_Picking[1] := BarcodeReader_Picking1.Done;

// NETWORK 14
BarcodeReader_Picking2B(
    Enable := bFl_RunningMachinePicking,
    Trigger := bFl_TriggerBarcode,
    InputBarcode := InputOutput_GVL.xIn_BarcodeReader_Picking2B,
    Enable_Out => InputOutput_GVL.xOut_BarcodeReader_Picking2B.TriggerEnable,
    TriggerBarcode => InputOutput_GVL.xOut_BarcodeReader_Picking2B.Trigger,
    AckResultBarcode => InputOutput_GVL.xOut_BarcodeReader_Picking2B.ResultsAck,
    GoodRead => bFl_GoodRead_Barcode_Picking[2],
    BadRead => bFl_BadRead_Barcode_Picking[2],
    Data => DataBarcode_Picking2,
    Error => Barcode2_Error); // DM_Connect
bFl_DoneRead_Barcode_Picking[2] := BarcodeReader_Picking2B.Done;

// NETWORK 15
BarcodeReader_Picking3B(
    Enable := bFl_RunningMachinePicking,
    Trigger := bFl_TriggerBarcode,
    InputBarcode := InputOutput_GVL.xIn_BarcodeReader_Picking3B,
    Enable_Out => InputOutput_GVL.xOut_BarcodeReader_Picking3B.TriggerEnable,
    TriggerBarcode => InputOutput_GVL.xOut_BarcodeReader_Picking3B.Trigger,
    AckResultBarcode => InputOutput_GVL.xOut_BarcodeReader_Picking3B.ResultsAck,
    GoodRead => bFl_GoodRead_Barcode_Picking[3],
    BadRead => bFl_BadRead_Barcode_Picking[3],
    Data => DataBarcode_Picking3,
    Error => Barcode3_Error); // DM_Connect
bFl_DoneRead_Barcode_Picking[3] := BarcodeReader_Picking3B.Done;

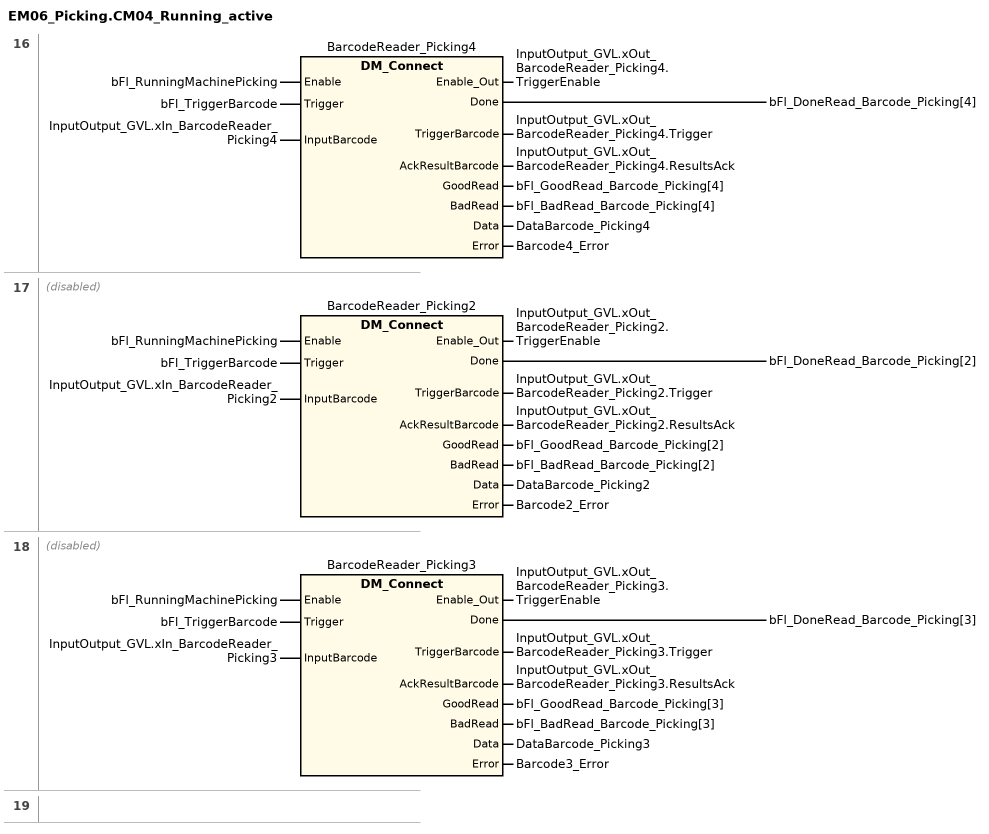
// NETWORK 16
BarcodeReader_Picking4(
    Enable := bFl_RunningMachinePicking,
    Trigger := bFl_TriggerBarcode,
    InputBarcode := InputOutput_GVL.xIn_BarcodeReader_Picking4,
    Enable_Out => InputOutput_GVL.xOut_BarcodeReader_Picking4.TriggerEnable,
    TriggerBarcode => InputOutput_GVL.xOut_BarcodeReader_Picking4.Trigger,
    AckResultBarcode => InputOutput_GVL.xOut_BarcodeReader_Picking4.ResultsAck,
    GoodRead => bFl_GoodRead_Barcode_Picking[4],
    BadRead => bFl_BadRead_Barcode_Picking[4],
    Data => DataBarcode_Picking4,
    Error => Barcode4_Error); // DM_Connect
bFl_DoneRead_Barcode_Picking[4] := BarcodeReader_Picking4.Done;

// NETWORK 17 (disabled)
// BarcodeReader_Picking2(
//     Enable := bFl_RunningMachinePicking,
//     Trigger := bFl_TriggerBarcode,
//     InputBarcode := InputOutput_GVL.xIn_BarcodeReader_Picking2,
//     Enable_Out => InputOutput_GVL.xOut_BarcodeReader_Picking2.TriggerEnable,
//     TriggerBarcode => InputOutput_GVL.xOut_BarcodeReader_Picking2.Trigger,
//     AckResultBarcode => InputOutput_GVL.xOut_BarcodeReader_Picking2.ResultsAck,
//     GoodRead => bFl_GoodRead_Barcode_Picking[2],
//     BadRead => bFl_BadRead_Barcode_Picking[2],
//     Data => DataBarcode_Picking2,
//     Error => Barcode2_Error); // DM_Connect
// bFl_DoneRead_Barcode_Picking[2] := BarcodeReader_Picking2.Done;

// NETWORK 18 (disabled)
// BarcodeReader_Picking3(
//     Enable := bFl_RunningMachinePicking,
//     Trigger := bFl_TriggerBarcode,
//     InputBarcode := InputOutput_GVL.xIn_BarcodeReader_Picking3,
//     Enable_Out => InputOutput_GVL.xOut_BarcodeReader_Picking3.TriggerEnable,
//     TriggerBarcode => InputOutput_GVL.xOut_BarcodeReader_Picking3.Trigger,
//     AckResultBarcode => InputOutput_GVL.xOut_BarcodeReader_Picking3.ResultsAck,
//     GoodRead => bFl_GoodRead_Barcode_Picking[3],
//     BadRead => bFl_BadRead_Barcode_Picking[3],
//     Data => DataBarcode_Picking3,
//     Error => Barcode3_Error); // DM_Connect
// bFl_DoneRead_Barcode_Picking[3] := BarcodeReader_Picking3.Done;

// NETWORK 19
END_ACTION

ACTION UP01_Backbone_active:
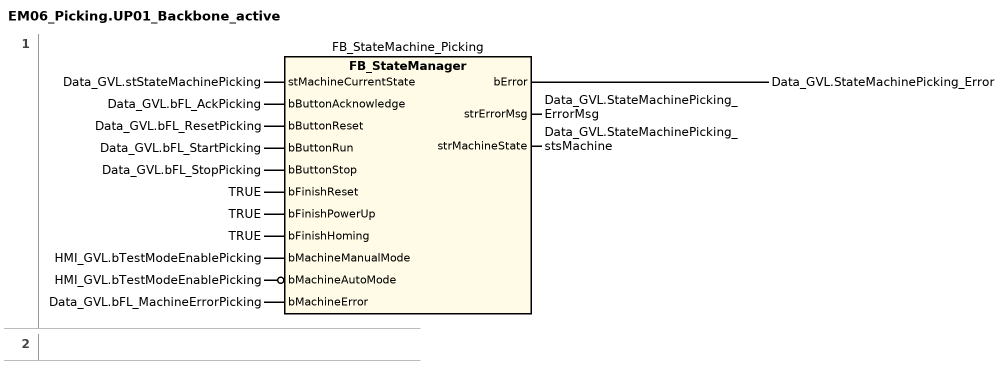
// NETWORK 1
FB_StateMachine_Picking(
    stMachineCurrentState := Data_GVL.stStateMachinePicking,
    bButtonAcknowledge := Data_GVL.bFL_AckPicking,
    bButtonReset := Data_GVL.bFL_ResetPicking,
    bButtonRun := Data_GVL.bFL_StartPicking,
    bButtonStop := Data_GVL.bFL_StopPicking,
    bFinishReset := TRUE,
    bFinishPowerUp := TRUE,
    bFinishHoming := TRUE,
    bMachineManualMode := HMI_GVL.bTestModeEnablePicking,
    bMachineAutoMode := NOT HMI_GVL.bTestModeEnablePicking,
    bMachineError := Data_GVL.bFL_MachineErrorPicking,
    strErrorMsg => Data_GVL.StateMachinePicking_ErrorMsg,
    strMachineState => Data_GVL.StateMachinePicking_stsMachine); // FB_StateManager
Data_GVL.StateMachinePicking_Error := FB_StateMachine_Picking.bError;

// NETWORK 2
END_ACTION

END_PROGRAM

// ---- POUs/Function_Block/General/Pneumatic_2Coil_Management.TcPOU
FUNCTION_BLOCK Pneumatic_2Coil_Management //V1.0
// Function block untuk mengolah faceplate dan watchdog pneumatic valve 2 coil
//	UDT dependencies:
	(*  
	1. stPneumatic2 v1.0 	*)

//	Changelog:
	(* 
	
	v1.0 [27.12.2021] Start development function block - Fabrilian Asali	
	v1.1 [24.05.2023] Add Pneumatic Name - Arif W*)	
	

VAR_INPUT
	bEnable						: BOOL;		
	bTriggerPneumaticRetract	: BOOL;
	bTriggerPneumaticAdvanced	: BOOL;
	bTriggerBoth				: BOOL;
	bReleaseBoth				: BOOL;
	bTestMode					: BOOL;
	bResetError					: BOOL;
	bBypassSensorRetract		: BOOL;
	bBypassSensorAdvanced		: BOOL;
	bBypassPreCheckSensor		: BOOL;
	xIn_SensorRetract			: BOOL;
	xIn_SensorAdvanced			: BOOL;
	TimerWatchdogRetract		: TIME := T#5S;
	TimerWatchdogAdvanced		: TIME := T#5S;
	TimerWatchdogPreRetract		: TIME := T#5S;
	TimerWatchdogPreAdvanced	: TIME := T#5S;
	TimerValve					: TIME := T#25MS;
	Name						: STRING;
END_VAR

VAR_OUTPUT
	bError						: BOOL;
	ErrorID						: INT;
	ErrorMsg					: STRING;
END_VAR

VAR_IN_OUT
	Pneumatic					: stPneumatic2;
END_VAR

VAR
	SeqIndex					: INT;
	SeqIndexAdv					: INT;
	SeqIndexRtc					: INT;
	InitSeqIndex				: INT;
	WatchdogTimer				: TON;
	ValveTimer					: TON;
	ValveTimerInit				: TON;
	bInit						: BOOL;
	PneuAdv						: R_TRIG;
	PneuRtc						: R_TRIG;
END_VAR
VAR // added by the converter: edge detectors and wires of the graphical bodies
    _w1 : BOOL;
    _rt1, _rt2, _rt3, _rt4 : R_TRIG;
END_VAR

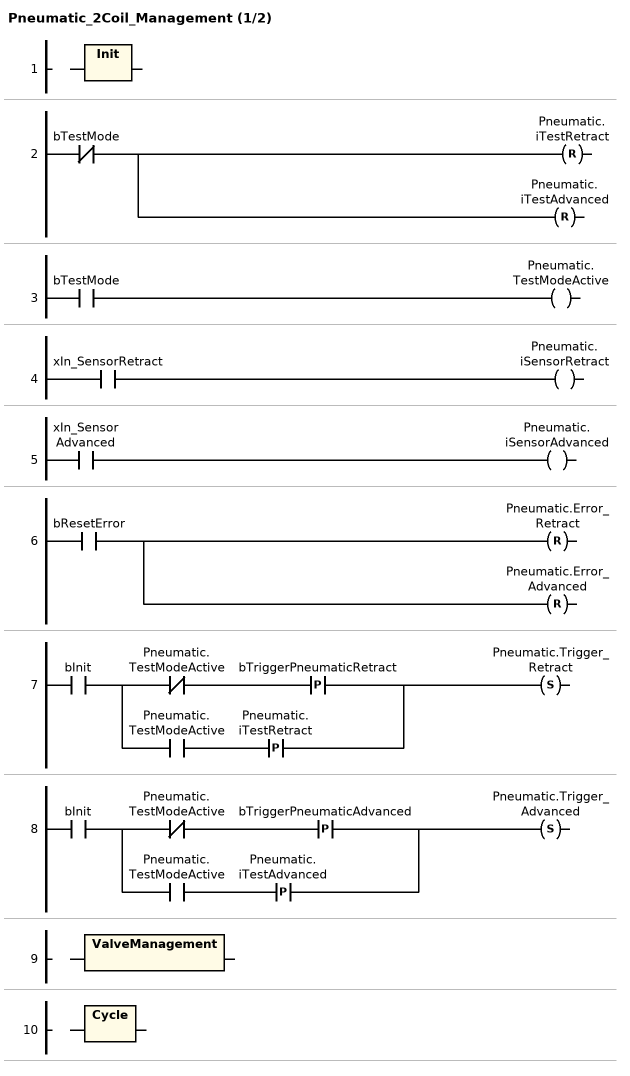
// NETWORK 1
Init();

// NETWORK 2
_w1 := NOT bTestMode;
Pneumatic.iTestRetract R= _w1;
Pneumatic.iTestAdvanced R= _w1;

// NETWORK 3
Pneumatic.TestModeActive := bTestMode;

// NETWORK 4
Pneumatic.iSensorRetract := xIn_SensorRetract;

// NETWORK 5
Pneumatic.iSensorAdvanced := xIn_SensorAdvanced;

// NETWORK 6
Pneumatic.Error_Retract R= bResetError;
Pneumatic.Error_Advanced R= bResetError;

// NETWORK 7
_rt1(CLK := bTriggerPneumaticRetract);
_rt2(CLK := Pneumatic.iTestRetract);
Pneumatic.Trigger_Retract S= bInit AND (NOT Pneumatic.TestModeActive AND _rt1.Q OR Pneumatic.TestModeActive AND _rt2.Q);

// NETWORK 8
_rt3(CLK := bTriggerPneumaticAdvanced);
_rt4(CLK := Pneumatic.iTestAdvanced);
Pneumatic.Trigger_Advanced S= bInit AND (NOT Pneumatic.TestModeActive AND _rt3.Q OR Pneumatic.TestModeActive AND _rt4.Q);

// NETWORK 9
ValveManagement();

// NETWORK 10
Cycle();

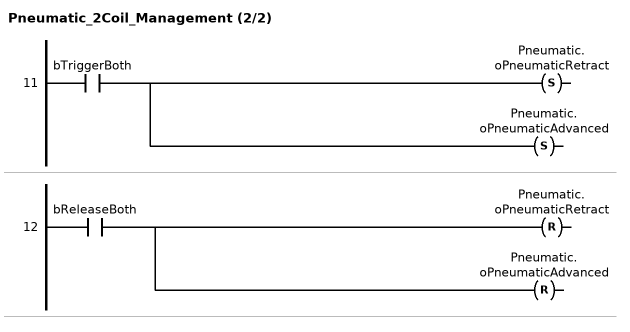
// NETWORK 11
Pneumatic.oPneumaticRetract S= bTriggerBoth;
Pneumatic.oPneumaticAdvanced S= bTriggerBoth;

// NETWORK 12
Pneumatic.oPneumaticRetract R= bReleaseBoth;
Pneumatic.oPneumaticAdvanced R= bReleaseBoth;

ACTION Cycle:
PneuAdv(CLK := Pneumatic.oPneumaticAdvanced AND Pneumatic.iSensorAdvanced);
IF PneuAdv.Q THEN
	Pneumatic.CyclePneuAdv	:= Pneumatic.CyclePneuAdv + 1;
END_IF


PneuRtc(CLK := Pneumatic.oPneumaticRetract AND Pneumatic.iSensorRetract);
IF PneuRtc.Q THEN
	Pneumatic.CyclePneuRtc	:= Pneumatic.CyclePneuRtc + 1;
END_IF
(*PneuAdv(CLK := Pneumatic.Trigger_Advanced);
CASE SeqIndexAdv OF
	0:
		IF PneuAdv.Q THEN
			Pneumatic.CyclePneuAdv	:= Pneumatic.CyclePneuAdv + 1;
			SeqIndexAdv				:= 1;
		END_IF
		
	1:
		IF NOT PneuAdv.Q THEN
			SeqIndexAdv				:= 0;
		END_IF
END_CASE

PneuRtc(CLK := Pneumatic.Trigger_Retract);
CASE SeqIndexRtc OF
	0:
		IF PneuRtc.Q THEN
			Pneumatic.CyclePneuRtc	:= Pneumatic.CyclePneuRtc + 1;
			SeqIndexRtc				:= 1;
		END_IF
		
	1:
		IF NOT PneuRtc.Q THEN
			SeqIndexRtc				:= 0;
		END_IF
END_CASE*)
END_ACTION

ACTION Init:
IF bResetError THEN
	bError			:= FALSE;
	InitSeqIndex	:= 0;
END_IF


IF bEnable AND NOT bInit THEN
	CASE InitSeqIndex OF
		0:
			IF xIn_SensorRetract THEN
				InitSeqIndex	:= 100;
			ELSIF xin_SensorAdvanced THEN
				InitSeqIndex	:= 200;
			ELSIF NOT xIn_SensorRetract AND NOT xIn_SensorAdvanced THEN
				InitSeqIndex	:= 300;
			ELSE
				ErrorID			:= 1;
				ErrorMsg		:= 'Both Sensor on at Init';
				InitSeqIndex	:= 999;
			END_IF
	
		100:
			Pneumatic.oPneumaticRetract 	:= TRUE;
			InitSeqIndex	:= 1000;
		
		200:
			Pneumatic.oPneumaticAdvanced	:= TRUE;
			InitSeqIndex	:= 1000;
		
		300:
			Pneumatic.oPneumaticRetract		:= TRUE;
			Pneumatic.oPneumaticAdvanced	:= TRUE;
			ValveTimerInit(In:= TRUE, PT:= TimerValve);
			IF ValveTimerInit.Q THEN
			    ValveTimerInit(In:=FALSE);
				Pneumatic.oPneumaticAdvanced := FALSE;
				Pneumatic.oPneumaticRetract := FALSE;
				InitSeqIndex := 1000;
			END_IF;
		
		999:
			bError	:= TRUE;
		
		1000:
			bInit	:= TRUE;
		
	END_CASE
END_IF
END_ACTION

ACTION ValveManagement:

IF bResetError THEN
	bError		:= FALSE;
	ErrorID		:= 0;
	ErrorMsg	:= '';
	SeqIndex	:= 0;
END_IF

IF bEnable AND bInit AND NOT bError THEN
	CASE SeqIndex OF
		0:
			IF Pneumatic.Trigger_Retract THEN
				SeqIndex	:= 100;
			ELSIF Pneumatic.Trigger_Advanced THEN
				SeqIndex	:= 200;
			END_IF
			
		100:
			Pneumatic.Trigger_Retract	:= FALSE;
			IF NOT bBypassPreCheckSensor THEN
				WatchdogTimer(In:= TRUE, PT:= TimerWatchdogPreRetract);
				IF Pneumatic.iSensorAdvanced THEN
					WatchdogTimer(In:= FALSE);
					SeqIndex	:= 105;
				ELSIF WatchdogTimer.Q THEN
					WatchdogTimer(In:= FALSE);
					Pneumatic.Error_Retract := TRUE;
					ErrorID					:= 10;
					ErrorMsg				:= CONCAT(Name,'Error PreCheck Retract');
					SeqIndex	:= 999;
				END_IF
			ELSE
				SeqIndex	:= 105;
			END_IF
	
		105:	
			Pneumatic.oPneumaticRetract		:= TRUE;
			Pneumatic.oPneumaticAdvanced	:= TRUE;
			ValveTimer(In:= TRUE, PT:= TimerValve);
			IF ValveTimer.Q THEN
				ValveTimer(In:= FALSE);
				Pneumatic.oPneumaticAdvanced	:= FALSE;
				SeqIndex	:= 110;
			END_IF
			
		110:
			IF NOT bBypassSensorRetract THEN
				WatchdogTimer(In:= TRUE, PT:= TimerWatchdogRetract);
				IF Pneumatic.iSensorRetract THEN
					WatchdogTimer(In:= FALSE);
					SeqIndex	:= 0;
				ELSIF WatchdogTimer.Q THEN
					WatchdogTimer(In:= FALSE);
					Pneumatic.Error_Retract := TRUE;
					ErrorID					:= 11;
					ErrorMsg				:= CONCAT(Name,'Error Watchdog Retract');
				END_IF
			ELSE
				SeqIndex	:= 0;
			END_IF
		
			
		200:
			Pneumatic.Trigger_Advanced	:= FALSE;
			IF NOT bBypassPreCheckSensor THEN
				WatchdogTimer(In:= TRUE, PT:= TimerWatchdogPreAdvanced);
				IF Pneumatic.iSensorRetract THEN
					WatchdogTimer(In:= FALSE);
					SeqIndex	:= 210;
				ELSIF WatchdogTimer.Q THEN
					WatchdogTimer(In:= FALSE);
					Pneumatic.Error_Advanced := TRUE;
					ErrorID					:= 20;
					ErrorMsg				:= CONCAT(Name,'Error PreCheck Advanced');
					SeqIndex	:= 999;
				END_IF
			ELSE
				SeqIndex	:= 205;
			END_IF				
		
		205:
			Pneumatic.oPneumaticRetract		:= TRUE;
			Pneumatic.oPneumaticAdvanced	:= TRUE;
			ValveTimer(In:= TRUE, PT:= TimerValve);
			IF ValveTimer.Q THEN
				Pneumatic.oPneumaticRetract	:= FALSE;
				SeqIndex	:= 210;
			END_IF	
			
		210:
			IF NOT bBypassSensorAdvanced THEN
				WatchdogTimer(In:= TRUE, PT:= TimerWatchdogAdvanced);
				IF Pneumatic.iSensorAdvanced THEN
					WatchdogTimer(In:= FALSE);
					SeqIndex	:= 0;
				ELSIF WatchdogTimer.Q THEN
					WatchdogTimer(In:= FALSE);
					Pneumatic.Error_Advanced := TRUE;
					ErrorID					:= 21;
					ErrorMsg				:= CONCAT(Name,'Error Watchdog Advanced');
				END_IF
			ELSE
				SeqIndex	:= 0;
			END_IF					
	
		999:
			bError	:= TRUE;	
	
	
	END_CASE
	
ELSE
	SeqIndex	:= 0;
	WatchdogTimer(IN:= FALSE);
END_IF
END_ACTION

END_FUNCTION_BLOCK

// ---- POUs/Function_Block/General/Pneumatic_1Coil_Management.TcPOU
FUNCTION_BLOCK Pneumatic_1Coil_Management
// Function block untuk mengolah faceplate dan watchdog pneumatic valve 1 coil
//	UDT dependencies:
	(*  
	1. stPneumatic v1.0 	*)

//	Changelog:
	(* 
	v1.0 [27.12.2021] Start development function block - Fabrilian Asali	*)	

VAR_INPUT
	bEnable						: BOOL;		
	bTriggerPneumatic			: BOOL;
	bTestMode					: BOOL;
	bResetError					: BOOL;
	bBypassSensorRetract		: BOOL;
	bBypassSensorAdvanced		: BOOL;
	bBypassPreCheckSensor		: BOOL;
	xIn_SensorRetract			: BOOL;
	xIn_SensorAdvanced			: BOOL;
	TimerBypassSensorRetract	: TIME := T#5S;
	TimerBypassSensorAdvanced	: TIME := T#5S;
	TimerWatchdogRetract		: TIME := T#5S;
	TimerWatchdogAdvanced		: TIME := T#5S;
	TimerWatchdogPreRetract		: TIME := T#5S;
	TimerWatchdogPreAdvanced	: TIME := T#5S;
END_VAR

VAR_OUTPUT
	bError						: BOOL;
	ErrorID						: INT;
	ErrorMsg					: STRING;
END_VAR

VAR_IN_OUT
	Pneumatic					: stPneumatic1;
END_VAR

VAR
	SeqIndex					: INT;
	WatchdogTimer				: TON;
	bTrig_Output				: BOOL;
	PneuAdv						: R_TRIG;
	TimerBypass					: TON;
END_VAR
VAR // added by the converter: edge detectors and wires of the graphical bodies
    _rt1 : R_TRIG;
END_VAR

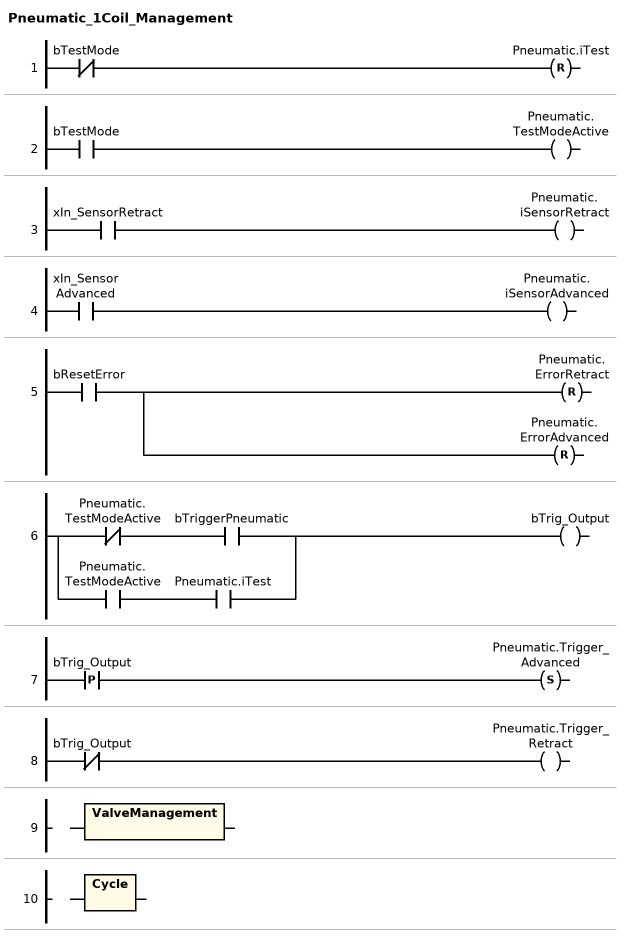
// NETWORK 1
Pneumatic.iTest R= NOT bTestMode;

// NETWORK 2
Pneumatic.TestModeActive := bTestMode;

// NETWORK 3
Pneumatic.iSensorRetract := xIn_SensorRetract;

// NETWORK 4
Pneumatic.iSensorAdvanced := xIn_SensorAdvanced;

// NETWORK 5
Pneumatic.ErrorRetract R= bResetError;
Pneumatic.ErrorAdvanced R= bResetError;

// NETWORK 6
bTrig_Output := NOT Pneumatic.TestModeActive AND bTriggerPneumatic OR Pneumatic.TestModeActive AND Pneumatic.iTest;

// NETWORK 7
_rt1(CLK := bTrig_Output);
Pneumatic.Trigger_Advanced S= _rt1.Q;

// NETWORK 8
Pneumatic.Trigger_Retract := NOT bTrig_Output;

// NETWORK 9
ValveManagement();

// NETWORK 10
Cycle();

ACTION Cycle:
PneuAdv (Clk := Pneumatic.oPneumatic);
IF PneuAdv.Q THEN
	Pneumatic.CyclePneu	:= Pneumatic.CyclePneu + 1;
END_IF
END_ACTION

ACTION ValveManagement:
IF bResetError THEN
	SeqIndex	:= 0;
	ErrorID		:= 0;
	ErrorMsg	:= '';
	bError		:= FALSE;
END_IF;

IF (bEnable OR Pneumatic.TestModeActive ) AND NOT bError THEN
	CASE SeqIndex OF
		0:
			WatchdogTimer(In:= FALSE);
			IF Pneumatic.Trigger_Retract AND NOT Pneumatic.FBDone_Retract THEN
				Pneumatic.FBDone_Retract:=FALSE;
				Pneumatic.FBDone_Advanced:=FALSE;
				SeqIndex	:= 100;
			ELSIF Pneumatic.Trigger_Advanced THEN
				Pneumatic.FBDone_Retract:=FALSE;
				Pneumatic.FBDone_Advanced:=FALSE;
				SeqIndex	:= 200;
			END_IF;
		
		100:
			Pneumatic.Trigger_Retract	:= FALSE;
			IF NOT bBypassPreCheckSensor THEN
				WatchdogTimer(In:= TRUE, PT:= TimerWatchdogPreRetract);
				IF Pneumatic.iSensorAdvanced THEN
					WatchdogTimer(In:= FALSE);
					SeqIndex	:= 110;
				ELSIF WatchdogTimer.Q THEN
					WatchdogTimer(In:= FALSE);
					Pneumatic.ErrorRetract := TRUE;
					ErrorID					:= 10;
					ErrorMsg				:= 'Error PreCheck Retract';
					SeqIndex	:= 999;
				END_IF;
			ELSE
				SeqIndex	:= 110;
			END_IF;
	
		110:
			Pneumatic.oPneumatic := FALSE;
			IF NOT bBypassSensorRetract THEN
				WatchdogTimer(In:= TRUE, PT:= TimerWatchdogRetract);
				IF Pneumatic.iSensorRetract THEN
					Pneumatic.FBDone_Retract:=TRUE;
					WatchdogTimer(In:= FALSE);
					SeqIndex	:= 0;
				ELSIF WatchdogTimer.Q THEN
					WatchdogTimer(In:= FALSE);
					Pneumatic.ErrorRetract := TRUE;
					ErrorID					:= 11;
					ErrorMsg				:= 'Error Watchdog Retract';
				END_IF;
			ELSE
				TimerBypass(In:= TRUE, PT:= TimerBypassSensorRetract);
				IF TimerBypass.Q THEN
					Pneumatic.FBDone_Retract:=TRUE;
					TimerBypass(In:= FALSE);
					SeqIndex	:= 0;
				END_IF;
			END_IF;
			
		200:
			Pneumatic.Trigger_Advanced	:= FALSE;
			IF NOT bBypassPreCheckSensor THEN
				WatchdogTimer(In:= TRUE, PT:= TimerWatchdogPreAdvanced);
				IF Pneumatic.iSensorRetract THEN
					WatchdogTimer(In:= FALSE);
					SeqIndex	:= 210;
				ELSIF WatchdogTimer.Q THEN
					WatchdogTimer(In:= FALSE);
					Pneumatic.ErrorAdvanced := TRUE;
					ErrorID					:= 20;
					ErrorMsg				:= 'Error PreCheck Advanced';
					SeqIndex	:= 999;
				END_IF;
			ELSE
				SeqIndex	:= 210;
			END_IF;				
		
		210:
			Pneumatic.oPneumatic := TRUE;
			IF NOT bBypassSensorAdvanced THEN
				WatchdogTimer(In:= TRUE, PT:= TimerWatchdogAdvanced);
				IF Pneumatic.iSensorAdvanced THEN
					Pneumatic.FBDone_Advanced:=TRUE;
					WatchdogTimer(In:= FALSE);
					SeqIndex	:= 0;
				ELSIF WatchdogTimer.Q THEN
					WatchdogTimer(In:= FALSE);
					Pneumatic.ErrorAdvanced := TRUE;
					ErrorID					:= 21;
					ErrorMsg				:= 'Error Watchdog Advanced';
				END_IF;
			ELSE
				TimerBypass(In:= TRUE, PT:= TimerBypassSensorAdvanced);
				IF TimerBypass.Q THEN
					Pneumatic.FBDone_Advanced:=TRUE;
					TimerBypass(In:= FALSE);
					SeqIndex	:= 0;
				END_IF;
				
			END_IF	;				
	
		999:
			bError	:= TRUE;	
			
	END_CASE;
ELSE
	IF bError OR Pneumatic.TestModeActive THEN
		SeqIndex := 0;
	END_IF;
	WatchdogTimer(IN:= FALSE);
	Pneumatic.Trigger_Advanced	:= FALSE;
	Pneumatic.Trigger_Retract	:= FALSE;
	Pneumatic.FBDone_Retract	:= FALSE;
	Pneumatic.FBDone_Advanced	:= FALSE;
END_IF;
END_ACTION

END_FUNCTION_BLOCK

// ---- POUs/Function_Block/Robot/FB_Picking.TcPOU
FUNCTION_BLOCK FB_Picking
VAR_INPUT
	Enable				: BOOL;
	bSensor1			: BOOL;
	bSensor2			: BOOL;
	bSensor3			: BOOL;
	bSensor4			: BOOL;
	StsCentering_Rtc	: BOOL;
	StsGapMaker_Rtc		: BOOL;
	StsGapMaker_Adv		: BOOL;
	bPickDone			: BOOL;
	Sts_Motor			: BOOL;
	BarcodeChecked		: BOOL;
	iRotate				: BOOL;
	iRotateInt			: USINT;
	BarcodePlace		: INT;
	Tmr_Check			: TIME;
	Tmr_Centering		: TIME;
	
END_VAR
VAR_OUTPUT
	PickReady			: BOOL;
	TrigBarcode			: BOOL;
	Sts_Busy			: BOOL;
	Motor_ON			: BOOL;
	Centering			: BOOL;
	GapMaker_Rtc		: BOOL;
	GapMaker_Adv		: BOOL;
	BigBox				: BOOL;
	SmallBox			: BOOL;
	oRotate				: BOOL;
	oRotateInt			: USINT;
	BoxType				: USINT;
	PickLine			: INT;
	CurrentJob			: STRING;
	SeqIndex			: INT;
END_VAR

VAR
	Sequence			: INT;
	DataTimer			: TON;
	Timeout				: TON;
END_VAR

IF Enable THEN
    CASE Sequence OF
        0:      (* Check Pneumatic Centering And GapMaker *)
			CurrentJob	:='Check Pneumatic Centering And GapMaker';
			Motor_ON	:= FALSE;
			GapMaker_Rtc:= TRUE;
			Centering	:= FALSE;
			IF StsCentering_Rtc AND StsGapMaker_Rtc THEN
				DataTimer(IN:= TRUE, PT:=T#100MS);
				IF DataTimer.Q THEN
					DataTimer(IN:= FALSE);
					GapMaker_Rtc:= FALSE;
					Sequence	:= 5;
				END_IF
			END_IF
			
		5:		(* Motor On *)
			CurrentJob	:='Motor On';
			Motor_ON	:= TRUE;
			IF bSensor1 AND bSensor2 THEN
				DataTimer(IN:= TRUE, PT:=Tmr_Check);
				IF DataTimer.Q THEN
					DataTimer(IN:= FALSE);
					Sequence	:= 20;
				END_IF
			ELSE
				DataTimer(IN:= FALSE);
				Sequence		:= 10;
			END_IF
			
		10:      (* Pneumatic GapMaker Advanced *)
			CurrentJob	:='Pneumatic GapMaker Advanced';
			GapMaker_Adv:= TRUE;
			IF StsGapMaker_Adv THEN
				DataTimer(IN:= TRUE, PT:=T#100MS);
				IF DataTimer.Q THEN
					DataTimer(IN:= FALSE);
					GapMaker_Adv:= FALSE;
					Sequence	:= 15;
				END_IF
			END_IF
			
		15:		(* Check Sensor *)
			CurrentJob	:='Check Sensor';
			Sts_Busy	:= FALSE;
			IF bSensor1 THEN
				Sts_Busy	:= TRUE;
				DataTimer(IN:= TRUE, PT:=Tmr_Check);
				IF DataTimer.Q THEN
					DataTimer(IN:= FALSE);
					Sequence	:= 20;
				END_IF
			END_IF
			
					
		20:		(* Pneumatic GapMaker Retract *)
			CurrentJob	:='Pneumatic GapMaker Retract';
			GapMaker_Rtc:= TRUE;
			Sts_Busy	:= TRUE;
			IF bSensor2 AND StsGapMaker_Rtc THEN
				DataTimer(IN:= TRUE, PT:=Tmr_Check);
				IF DataTimer.Q THEN
					DataTimer(IN:= FALSE);
					Motor_ON	:= FALSE;
					GapMaker_Rtc:= FALSE;
					IF NOT Sts_Motor THEN
						Sequence	:= 30;
					END_IF
				END_IF
			ELSIF NOT bSensor1 AND NOT bSensor2 THEN
				Timeout(IN:=TRUE, PT:=T#3S);
				IF Timeout.Q THEN
					Timeout(IN:=FALSE);
					BigBox		:= FALSE;
					SmallBox	:= FALSE;
					PickReady	:= FALSE;
					TrigBarcode	:= FALSE;
					oRotate		:= FALSE;
					oRotateInt	:= 0;
					BoxType		:= 0;
					PickLine	:= 0;
					Sequence	:= 0;
				END_IF
			END_IF
			
		30:		(* Centering Box *)
			CurrentJob	:='Centering Box';
			DataTimer(IN:= TRUE, PT:=Tmr_Centering);
			IF DataTimer.Q THEN
				Centering	:= FALSE;
			ELSE
				Centering	:= TRUE;
			END_IF
			IF StsCentering_Rtc AND DataTimer.Q THEN
				DataTimer(IN:= FALSE);
				Sequence	:= 40;
			END_IF
			
		40:		(* Trigger Barcode Reader *)
			CurrentJob	:='Trigger Barcode Reader';
			TrigBarcode	:= TRUE;
			IF bSensor3 THEN
				BigBox	:= TRUE;
			ELSE
				BigBox	:= FALSE;
			END_IF
			IF NOT bSensor4 AND NOT bSensor3 THEN
				SmallBox:= TRUE;
			ELSE
				SmallBox:= FALSE;
			END_IF
			
			IF bSensor3 THEN
				BoxType	:= 3; //Standard Case
			ELSIF bSensor2 AND NOT bSensor3 THEN
				BoxType	:= 2; //Small Case
			ELSE
				BoxType	:= 1; //LU 18
			END_IF
			IF BarcodeChecked THEN
				Sequence	:= 45;
			ELSIF NOT bSensor1 AND NOT bSensor2 THEN
				Timeout(IN:=TRUE, PT:=T#3S);
				IF Timeout.Q THEN
					Timeout(IN:=FALSE);
					BigBox		:= FALSE;
					SmallBox	:= FALSE;
					PickReady	:= FALSE;
					TrigBarcode	:= FALSE;
					oRotate		:= FALSE;
					oRotateInt	:= 0;
					BoxType		:= 0;
					PickLine	:= 0;
					Sequence	:= 0;
				END_IF
			END_IF
			
		45:
			CurrentJob	:='Check...';
			PickLine	:= BarcodePlace;
			oRotate		:= iRotate;
			oRotateInt	:= iRotateInt;
			DataTimer(IN:=TRUE, PT:=T#10MS);
			IF DataTimer.Q THEN
				Sequence	:= 50;
			END_IF
			
			
		50:		(* Pick Ready *)
			CurrentJob	:='Pick Ready';
			PickReady	:= TRUE;
			IF bPickDone THEN
				Sequence	:= 60;
			ELSIF NOT bSensor1 AND NOT bSensor2 THEN
				DataTimer(IN:=TRUE, PT:=T#3S);
				IF DataTimer.Q THEN
					DataTimer(IN:=FALSE);
					BigBox		:= FALSE;
					SmallBox	:= FALSE;
					PickReady	:= FALSE;
					TrigBarcode	:= FALSE;
					oRotate		:= FALSE;
					oRotateInt	:= 0;
					BoxType		:= 0;
					PickLine	:= 0;
					Sequence	:= 0;
				END_IF
			END_IF
			
		60:
			IF NOT bPickDone THEN
				BigBox		:= FALSE;
				SmallBox	:= FALSE;
				PickReady	:= FALSE;
				TrigBarcode	:= FALSE;
				oRotate		:= FALSE;
				oRotateInt	:= 0;
				BoxType		:= 0;
				PickLine	:= 0;
				Sequence	:= 0;
			ELSIF NOT bSensor1 AND NOT bSensor2 THEN
				DataTimer(IN:=TRUE, PT:=T#3S);
				IF DataTimer.Q THEN
					DataTimer(IN:=FALSE);
					BigBox		:= FALSE;
					SmallBox	:= FALSE;
					PickReady	:= FALSE;
					TrigBarcode	:= FALSE;
					oRotate		:= FALSE;
					oRotateInt	:= 0;
					BoxType		:= 0;
					PickLine	:= 0;
					Sequence	:= 0;
				END_IF
			END_IF
			
    END_CASE;
ELSE
   Sequence 	:= 0;
   oRotateInt	:= 0;
   BoxType		:= 0;
   CurrentJob	:='Machine Stopped';
   Sts_Busy		:= TRUE;
   BigBox		:= FALSE;
   SmallBox		:= FALSE;
   PickReady 	:= FALSE;
   Motor_ON 	:= FALSE;
   Centering	:= FALSE;
   GapMaker_Rtc	:= FALSE;
   GapMaker_Adv	:= FALSE;
   TrigBarcode	:= FALSE;
   DataTimer(IN := FALSE);
END_IF;

SeqIndex	:= Sequence;

END_FUNCTION_BLOCK

// ---- POUs/Function_Block/Robot/FB_BarcodeInspection.TcPOU
FUNCTION_BLOCK FB_BarcodeInspection
VAR_INPUT
	bEnable				: BOOL;
	bTrigger			: BOOL;
	bBypassFGHS			: BOOL;
	bBarcodeGood		: ARRAY [1..4] OF BOOL;
	bBarcodeBad			: ARRAY [1..4] OF BOOL;
	bDoneRead			: ARRAY [1..4] OF BOOL;
	BarcodeData1		: STRING;
	BarcodeData2		: STRING;
	BarcodeData3		: STRING;
	BarcodeData4		: STRING;
	bPalletReady		: ARRAY [1..4] OF BOOL;
	bResetCounter		: BOOL;
END_VAR
VAR_OUTPUT
	bBarcodeChecked		: BOOL;
	BarcodeResult		: STRING;
	iPlacingLine		: INT;
	bReject				: BOOL;
	bProductFound		: ARRAY [1..4] OF BOOL;
	RejectID			: INT;
	RejectMsg			: STRING;
END_VAR
VAR_OUTPUT PERSISTENT
	CountReject			: UINT;
END_VAR
VAR_IN_OUT
	ar_ProductInfo		: ARRAY [1..4] OF stProductInfo;
	PlannedEAN			: ARRAY [1..4] OF STRING;
	PlannedCodeVariant	: ARRAY [1..4] OF STRING;
END_VAR
VAR
	Sequence			: INT;
	DoneCheck			: BOOL;
	BarcodeEAN			: STRING;
	CodeVariant			: STRING;
	BarcodeLinkUp		: STRING;
	TimeOut				: TON;
	NotFound			: BOOL;
	i					: INT;
	Index				: INT;
END_VAR

IF bResetCounter THEN
	CountReject := 0;
END_IF

IF bEnable THEN
	
	(*----Check Barcode -----*)
	CASE Sequence OF
		0:	
			IF bTrigger THEN
				DoneCheck		:= FALSE;
				bBarcodeChecked	:= FALSE;
				bReject			:= FALSE;
				iPlacingLine	:= 0;
				RejectID		:= 0;
				RejectMsg		:= '';
				BarcodeResult	:= '';
				BarcodeEAN		:= '';
				CodeVariant		:= '';
				BarcodeLinkUp	:= '';
				Sequence		:= 10;
			END_IF
			
		10:
			TimeOut(IN:=TRUE, PT:=T#5S);
			IF bBarcodeGood[1] AND bDoneRead[1] THEN
				BarcodeResult 	:= BarcodeData1;
				Sequence		:= 11;
			ELSIF bBarcodeGood[2] AND bDoneRead[2] THEN
				BarcodeResult 	:= BarcodeData2;
				Sequence		:= 11;
			ELSIF bBarcodeGood[3] AND bDoneRead[3] THEN
				BarcodeResult 	:= BarcodeData3;
				Sequence		:= 11;
			ELSIF bBarcodeGood[4] AND bDoneRead[4] THEN
				BarcodeResult 	:= BarcodeData4;
				Sequence		:= 11;
			ELSIF (bBarcodeBad[1] AND bBarcodeBad[2] AND bBarcodeBad[3] AND bBarcodeBad[4]) OR TimeOut.Q  THEN //
				TimeOut(IN:=FALSE); 
				RejectID		:= 1;
				RejectMsg		:= 'Reject Bad Read Barcode';
				Sequence		:= 999; 
			END_IF
			
		11:	(* Split Barcode *)
			BarcodeEAN		:= DELETE(DELETE(BarcodeResult,3,0),24,15);
			CodeVariant		:= DELETE(DELETE(BarcodeResult,19,0),20,3);
			BarcodeLinkUp	:= DELETE(DELETE(BarcodeResult,33,0),6,3);
			Sequence		:= 12;
			
		12: (* Check EAN *)
			FOR i := 1 TO 4 BY 1 DO
				IF PlannedEAN[i] <> '' AND BarcodeEAN = PlannedEAN[i] AND PlannedEAN[i] <> ar_ProductInfo[i].EANVariant THEN
					ar_ProductInfo[i].EANVariant	:= PlannedEAN[i];
					bProductFound[i]				:= TRUE;
					Sequence						:= 20;
					EXIT;
				END_IF
			END_FOR
			
			IF i > 4 THEN
				i 				:= 0;
				Sequence		:= 20;
			END_IF
			
		20:	
			FOR i := 1 TO 4 BY 1 DO
				IF BarcodeLinkUp = ar_ProductInfo[i].LinkUpSource  AND BarcodeEAN = ar_ProductInfo[i].EANVariant THEN //AND CodeVariant = ar_ProductInfo[i].CodeVariant
					iPlacingLine	 		:= i;
					Sequence				:= 21;
				EXIT;
				END_IF;
			END_FOR;	
			IF i > 4 THEN
				bBarcodeChecked	:= FALSE;
				NotFound		:= TRUE;
				RejectID		:= 2;
				RejectMsg		:= 'Barcode Result Not Matched Any References';
				Sequence		:= 999;
			END_IF;
			
		21:
			IF CodeVariant <> ar_ProductInfo[iPlacingLine].CodeVariant THEN
				ar_ProductInfo[iPlacingLine].CodeVariant	:= CodeVariant;
				bProductFound[iPlacingLine]					:= TRUE;
				Sequence									:= 30;
			ELSE
				Sequence									:= 30;
			END_IF
			
		30:
			IF bPalletReady[iPlacingLine] THEN
				TimeOut(IN:=FALSE);
				bBarcodeChecked	:=	TRUE;
				Sequence		:=	1000;	
			ELSE
				TimeOut(IN:=TRUE, PT:=T#30S);
				IF TimeOut.Q THEN
				TimeOut(IN:=FALSE);
				RejectID		:= 3;
				RejectMsg		:= 'Reject Placing Not Ready';
				Sequence		:= 999;
				END_IF
			END_IF
			
		999:
			TimeOut(IN:=FALSE);
			iPlacingLine	:= 0;
			bBarcodeChecked	:=	TRUE;
			bReject 		:=	TRUE;
			CountReject		:= 	CountReject + 1;
			Sequence		:=	1000;	
	
		1000:
			DoneCheck	:= TRUE;
			IF NOT bTrigger THEN
				bProductFound[1]	:= FALSE;	
				bProductFound[2]	:= FALSE;
				bProductFound[3]	:= FALSE;
				bProductFound[4]	:= FALSE;
				NotFound			:= FALSE;
				bBarcodeChecked		:= FALSE;
				bReject				:= FALSE;
				Sequence			:= 0;
			END_IF
			
	END_CASE
	
	
ELSE
	TimeOut(IN:=FALSE);
	NotFound			:= FALSE;
	bBarcodeChecked		:= FALSE;
	bReject				:= FALSE;
	Sequence			:= 0;
	iPlacingLine		:= 0;
	i					:= 0;
END_IF

END_FUNCTION_BLOCK

// ---- POUs/Function_Block/Robot/DM_Connect.TcPOU
FUNCTION_BLOCK DM_Connect
VAR_INPUT
	Enable			: BOOL;
	Trigger			: BOOL;
	InputBarcode	: stDM_Input;
END_VAR


VAR_OUTPUT
	Enable_Out			: BOOL;
	Done				: BOOL;
	TriggerBarcode		: BOOL;
	AckResultBarcode	: BOOL;
	GoodRead			: BOOL;
	BadRead				: BOOL;
	Data				: STRING;
	Error				: BOOL;
END_VAR


VAR
	SeqIndex	: INT;
	DataTimer	: TON;
	BufferData	: ARRAY [0..MAX_STRING_LENGTH] OF BYTE;
	i			: DINT;
END_VAR

IF Enable THEN
	Enable_Out	:= TRUE;
	CASE SeqIndex OF
		0:
			IF Trigger THEN
				GoodRead:=FALSE;
				BadRead	:=FALSE;
				Done	:=FALSE;
				SeqIndex:=1;
			END_IF;
		1:
			IF InputBarcode.ResultsAvailable THEN
				AckResultBarcode:=TRUE;
				SeqIndex:=2;
			ELSE
				SeqIndex:=10;
			END_IF;
		2:
			IF NOT InputBarcode.ResultsAvailable THEN
				AckResultBarcode:=FALSE;
				SeqIndex:=10;
			END_IF;
		10:
			TriggerBarcode:=TRUE;
			IF InputBarcode.TriggerAck THEN
				DataTimer(IN:=FALSE);
				TriggerBarcode:=FALSE;
				SeqIndex:=20;
			ELSE
				DataTimer(IN:=TRUE,PT:=T#20S);
				IF DataTimer.Q THEN
					DataTimer(IN:=FALSE);
					SeqIndex:=1000;
				END_IF;
			END_IF;
		20:
			IF InputBarcode.ResultsAvailable THEN
				DataTimer(IN:=FALSE);
				SeqIndex:=30;
			ELSE
				DataTimer(IN:=TRUE,PT:=T#20S);
				IF DataTimer.Q THEN
					DataTimer(IN:=FALSE);
					SeqIndex:=1000;
				END_IF;
			END_IF;
		30:
			IF InputBarcode.ResultCode = 1 THEN
				SeqIndex:=100;
			ELSE
				SeqIndex:=110;
			END_IF;
		100:
			GoodRead:=TRUE;
			BadRead	:=FALSE;
			FOR i:=0 TO InputBarcode.ResultDataLength BY 1 DO
				BufferData[i]:=InputBarcode.ResultData[i];
			END_FOR
			Data:=BYTEARR_TO_MAXSTRING(BufferData);
			SeqIndex:=200;
		110:
			GoodRead	:=FALSE;
			BadRead		:=TRUE;
			Data		:='Not Read';
			DataTimer(IN:=FALSE);
			SeqIndex:=200;
		200:
			Done:=TRUE;
			IF NOT Trigger THEN
				DataTimer(IN:=TRUE,PT:=T#10MS);
				IF DataTimer.Q THEN
					DataTimer(IN:=FALSE);
					Done:=FALSE;
					SeqIndex:=210;
				END_IF
	
			END_IF;
		210:
			AckResultBarcode:=TRUE;
			IF NOT InputBarcode.ResultsAvailable THEN
				AckResultBarcode:=FALSE;
				SeqIndex:=0;
			END_IF;
		1000:
			Error:=TRUE;
			IF NOT Trigger THEN
				Error:=FALSE;
				TriggerBarcode:=FALSE;
				SeqIndex:=0;
			END_IF;
	END_CASE;
ELSE
	DataTimer(IN:=FALSE);
	Enable_Out		:= FALSE;
	AckResultBarcode:=FALSE;
	Error			:=FALSE;
	TriggerBarcode	:=FALSE;
	GoodRead		:=FALSE;
	BadRead			:=FALSE;
	Done			:=FALSE;
	SeqIndex		:=0;
END_IF;

END_FUNCTION_BLOCK

// ---- POUs/Function_Block/General/RejectMsgHandling.TcPOU
FUNCTION_BLOCK RejectMsgHandling
VAR_INPUT
	bReject			: BOOL;
	bRejectID		: INT;
	RejectType		: STRING;
	Counter			: UINT;
	RejectMsg		: STRING;
	Timestamp		: STRING;	
	bResetBuffer	: BOOL;
END_VAR
VAR_OUTPUT
END_VAR
VAR_IN_OUT
	dtRejectHistory	: ARRAY [1..20] OF stRejectData;
END_VAR
VAR
	i				: UINT;
	j				: UINT;
	LastIndex		: UINT;
	EmptyArray		: ARRAY [1..20] OF stRejectData;
	SeqIndex		: UINT;
	
END_VAR


	CASE SeqIndex OF
		0:
			IF bReject THEN
				SeqIndex	:= 5;	
			END_IF
			
		5:
			FOR i := 1 TO 20 BY 1 DO
			IF dtRejectHistory[i].Status = 0 THEN
				LastIndex	:= i;
				SeqIndex	:= 10;
				EXIT;
			END_IF
			END_FOR
				
			IF i > 20 THEN
				SeqIndex	:= 10;
			END_IF
			
			
		10:
			IF LastIndex > 1 THEN
				FOR j := LastIndex TO 2 BY -1 DO
					dtRejectHistory[j].Status		:=	dtRejectHistory[j-1].Status;
					dtRejectHistory[j].RejectID		:=	dtRejectHistory[j-1].RejectID;
					dtRejectHistory[j].RejectType	:=	dtRejectHistory[j-1].RejectType;
					dtRejectHistory[j].Counter		:=	dtRejectHistory[j-1].Counter;
					dtRejectHistory[j].RejectMsg	:=	dtRejectHistory[j-1].RejectMsg;
					dtRejectHistory[j].Timestamp	:=	dtRejectHistory[j-1].Timestamp;
				END_FOR
			END_IF
			
			//IF j >= LastIndex THEN
				SeqIndex	:= 20;
			//END_IF
			
		20:
				dtRejectHistory[1].Status			:=	1;
				dtRejectHistory[1].RejectID			:=	bRejectID;
				dtRejectHistory[1].RejectType		:=	RejectType;
				dtRejectHistory[1].Counter			:=	Counter+1;
				dtRejectHistory[1].RejectMsg		:=	RejectMsg;
				dtRejectHistory[1].Timestamp		:=	Timestamp;
				IF NOT bReject THEN
					i			:= 0;
					j			:= 0;
					SeqIndex	:= 0;
				END_IF
			
	END_CASE
	

IF bResetBuffer	THEN //OR LastIndex >= 20
	LastIndex		:= 0;
	i				:= 0;
	j				:= 0;
	SeqIndex		:= 0;
	dtRejectHistory	:= EmptyArray;
END_IF

END_FUNCTION_BLOCK

// ---- POUs/S00_System_Utilities/Module_Status.TcPOU
PROGRAM Module_Status
VAR
	BLINK_Check		: Blink;
	BLINK_Module	: Blink;
	Index			: INT;
	TimerModule		: ARRAY [1..10] OF TOF;
	Ethercat_Status : ARRAY [1..10] OF Ethercat_status;
	FB_SystemData	: SystemData;
	FB_CpuUsage		: TC_CpuUsage;
	FB_SysLatency	: TC_SysLatency;
	FB_UPS			: FB_S_UPS_CX51x0;
END_VAR

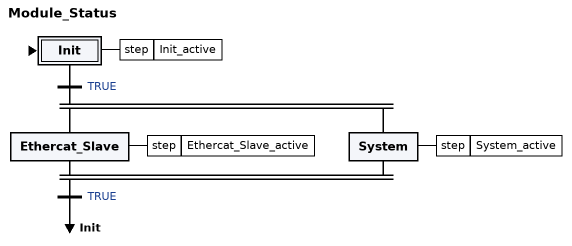
INITIAL_STEP Init:
    Init_active(N);  // step action
END_STEP
TRANSITION FROM Init TO (Ethercat_Slave, System)
    := TRUE;
END_TRANSITION
STEP Ethercat_Slave:
    Ethercat_Slave_active(N);  // step action
END_STEP
STEP System:
    System_active(N);  // step action
END_STEP
TRANSITION FROM (Ethercat_Slave, System) TO Init
    := TRUE;
END_TRANSITION

ACTION Ethercat_Slave_active:
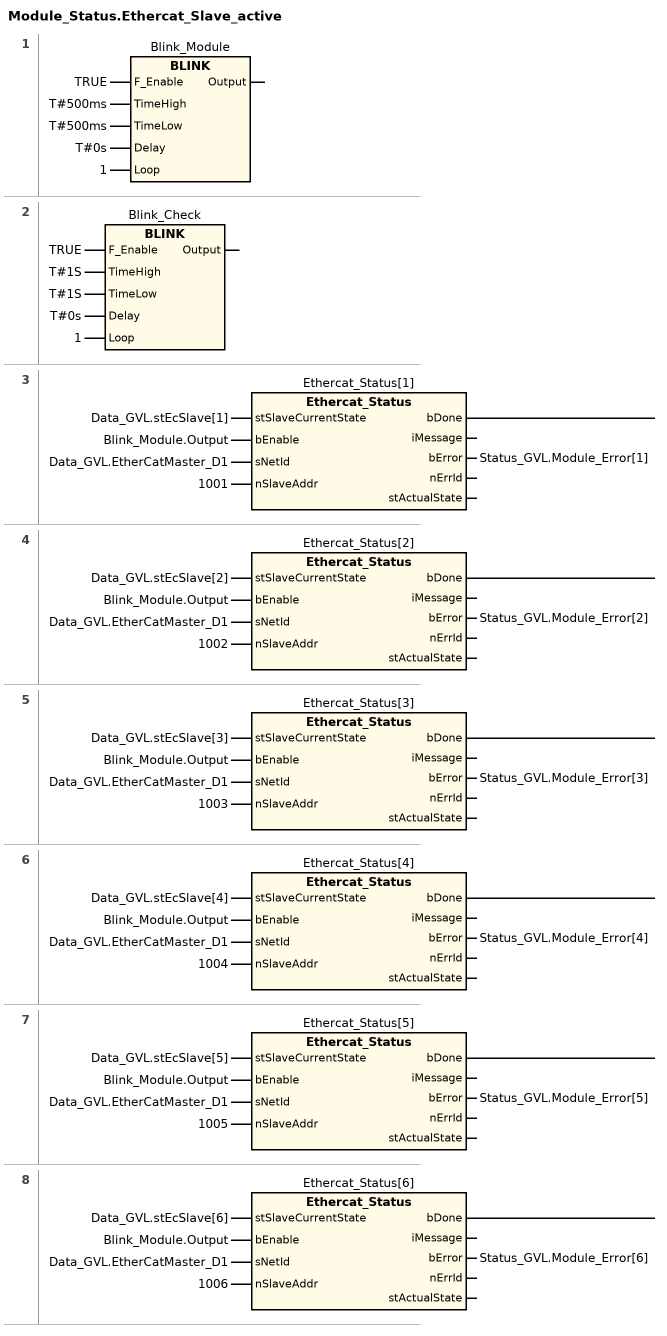
// NETWORK 1
Blink_Module(F_Enable := TRUE, TimeHigh := T#500ms, TimeLow := T#500ms, Delay := T#0s, Loop := 1); // BLINK

// NETWORK 2
Blink_Check(F_Enable := TRUE, TimeHigh := T#1S, TimeLow := T#1S, Delay := T#0s, Loop := 1); // BLINK

// NETWORK 3
Ethercat_Status[1](
    stSlaveCurrentState := Data_GVL.stEcSlave[1],
    bEnable := Blink_Module.Output,
    sNetId := Data_GVL.EtherCatMaster_D1,
    nSlaveAddr := 1001,
    bError => Status_GVL.Module_Error[1]); // Ethercat_Status

// NETWORK 4
Ethercat_Status[2](
    stSlaveCurrentState := Data_GVL.stEcSlave[2],
    bEnable := Blink_Module.Output,
    sNetId := Data_GVL.EtherCatMaster_D1,
    nSlaveAddr := 1002,
    bError => Status_GVL.Module_Error[2]); // Ethercat_Status

// NETWORK 5
Ethercat_Status[3](
    stSlaveCurrentState := Data_GVL.stEcSlave[3],
    bEnable := Blink_Module.Output,
    sNetId := Data_GVL.EtherCatMaster_D1,
    nSlaveAddr := 1003,
    bError => Status_GVL.Module_Error[3]); // Ethercat_Status

// NETWORK 6
Ethercat_Status[4](
    stSlaveCurrentState := Data_GVL.stEcSlave[4],
    bEnable := Blink_Module.Output,
    sNetId := Data_GVL.EtherCatMaster_D1,
    nSlaveAddr := 1004,
    bError => Status_GVL.Module_Error[4]); // Ethercat_Status

// NETWORK 7
Ethercat_Status[5](
    stSlaveCurrentState := Data_GVL.stEcSlave[5],
    bEnable := Blink_Module.Output,
    sNetId := Data_GVL.EtherCatMaster_D1,
    nSlaveAddr := 1005,
    bError => Status_GVL.Module_Error[5]); // Ethercat_Status

// NETWORK 8
Ethercat_Status[6](
    stSlaveCurrentState := Data_GVL.stEcSlave[6],
    bEnable := Blink_Module.Output,
    sNetId := Data_GVL.EtherCatMaster_D1,
    nSlaveAddr := 1006,
    bError => Status_GVL.Module_Error[6]); // Ethercat_Status

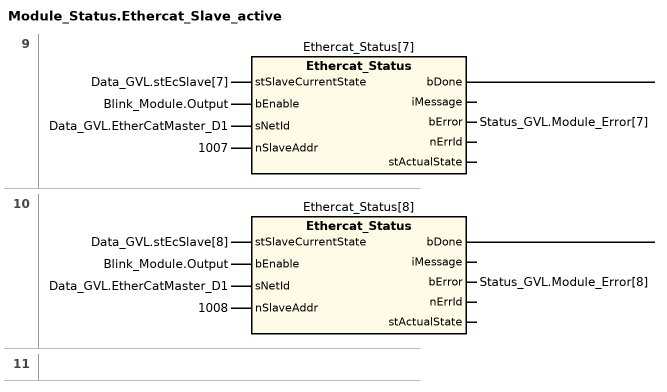
// NETWORK 9
Ethercat_Status[7](
    stSlaveCurrentState := Data_GVL.stEcSlave[7],
    bEnable := Blink_Module.Output,
    sNetId := Data_GVL.EtherCatMaster_D1,
    nSlaveAddr := 1007,
    bError => Status_GVL.Module_Error[7]); // Ethercat_Status

// NETWORK 10
Ethercat_Status[8](
    stSlaveCurrentState := Data_GVL.stEcSlave[8],
    bEnable := Blink_Module.Output,
    sNetId := Data_GVL.EtherCatMaster_D1,
    nSlaveAddr := 1008,
    bError => Status_GVL.Module_Error[8]); // Ethercat_Status

// NETWORK 11
END_ACTION

ACTION Init_active:
IF Blink_Check.Output THEN
	FOR Index := 1 TO 10 BY 1 DO
		TimerModule[Index](In:= Data_GVL.stEcSlave[Index].OP, PT:= T#2S);
		IF NOT TimerModule[Index].Q THEN 
			HMI_GVL.xOut_HMI_Status_EcSlave[Index] := FALSE;
		ELSE 
			HMI_GVL.xOut_HMI_Status_EcSlave[Index] := TRUE;
		END_IF
		
	END_FOR
ELSE
	Index := 1;
END_IF
END_ACTION

ACTION System_active:
